LIN {X 0,Y 382.363,Z 610.569,A -85,B 0,C 180,E1 -11975.801,E2 -11975.801} C_VEL
LIN {X 0,Y 382.259,Z 606.99,A -85,B 0,C 180,E1 -11977.393,E2 -11977.393} C_VEL
LIN {X 0,Y 382.264,Z 602.395,A -85,B 0,C 180,E1 -11978.989,E2 -11978.989} C_VEL
LIN {X 0,Y 382.468,Z 595.707,A -85,B 0,C 180,E1 -11980.855,E2 -11980.855} C_VEL
LIN {X 0,Y 382.818,Z 587.32,A -85,B 0,C 180,E1 -11982.726,E2 -11982.726} C_VEL
LIN {X 0,Y 383.476,Z 578.596,A -85,B 0,C 180,E1 -11984.323,E2 -11984.323} C_VEL
LIN {X 0,Y 384.358,Z 568.07,A -85,B 0,C 180,E1 -11985.917,E2 -11985.917} C_VEL
LIN {X 0,Y 385.396,Z 557.58,A -85,B 0,C 180,E1 -11987.236,E2 -11987.236} C_VEL
LIN {X 0,Y 386.433,Z 546.274,A -85,B 0,C 180,E1 -11988.42,E2 -11988.42} C_VEL
LIN {X 0,Y 387.509,Z 533.775,A -85,B 0,C 180,E1 -11989.493,E2 -11989.493} C_VEL
LIN {X 0,Y 387.828,Z 526.827,A -85,B 0,C 180,E1 -11990.006,E2 -11990.006} C_VEL
LIN {X 0,Y 386.566,Z 512.32,A -85,B 0,C 180,E1 -11990.954,E2 -11990.954} C_VEL
LIN {X 0,Y 384.765,Z 496.815,A -85,B 0,C 180,E1 -11991.736,E2 -11991.736} C_VEL
LIN {X 0,Y 383.032,Z 482.96,A -85,B 0,C 180,E1 -11992.27,E2 -11992.27} C_VEL
LIN {X 0,Y 383.628,Z 472.139,A -85,B 0,C 180,E1 -11995.499,E2 -11995.499} C_VEL
LIN {X 0,Y 384.429,Z 460.422,A -85,B 0,C 180,E1 -11999.048,E2 -11999.048} C_VEL
LIN {X 0,Y 385.201,Z 450.992,A -85,B 0,C 180,E1 -12001.943,E2 -12001.943} C_VEL
LIN {X 0,Y 386.105,Z 441.213,A -85,B 0,C 180,E1 -12005.005,E2 -12005.005} C_VEL
LIN {X 0,Y 387.399,Z 428.707,A -85,B 0,C 180,E1 -12009.008,E2 -12009.008} C_VEL
LIN {X 0,Y 387.577,Z 424.534,A -85,B 0,C 180,E1 -12010.395,E2 -12010.395} C_VEL
LIN {X 0,Y 386.394,Z 417.864,A -85,B 0,C 180,E1 -12012.764,E2 -12012.764} C_VEL
LIN {X 0,Y 384.278,Z 407.541,A -85,B 0,C 180,E1 -12016.612,E2 -12016.612} C_VEL
LIN {X 0,Y 383.036,Z 401.399,A -85,B 0,C 180,E1 -12019.079,E2 -12019.079} C_VEL
LIN {X 0,Y 382.99,Z 401.403,A -85,B 0,C 180,E1 -12022.731,E2 -12022.731} C_VEL
LIN {X 0,Y 383.008,Z 401.4,A -85,B 0,C 180,E1 -12025.659,E2 -12025.659} C_VEL
LIN {X 0,Y 382.977,Z 401.407,A -85,B 0,C 180,E1 -12029.081,E2 -12029.081} C_VEL
LIN {X 0,Y 383.047,Z 401.395,A -85,B 0,C 180,E1 -12032.698,E2 -12032.698} C_VEL
LIN {X 0,Y 383.023,Z 401.396,A -85,B 0,C 180,E1 -12036.192,E2 -12036.192} C_VEL
LIN {X 0,Y 383.045,Z 401.395,A -85,B 0,C 180,E1 -12039.598,E2 -12039.598} C_VEL
LIN {X 0,Y 383.094,Z 401.392,A -85,B 0,C 180,E1 -12042.931,E2 -12042.931} C_VEL
LIN {X 0,Y 383.115,Z 401.386,A -85,B 0,C 180,E1 -12046.463,E2 -12046.463} C_VEL
LIN {X 0,Y 383.13,Z 401.385,A -85,B 0,C 180,E1 -12049.43,E2 -12049.43} C_VEL
LIN {X 0,Y 383.262,Z 401.369,A -85,B 0,C 180,E1 -12052.625,E2 -12052.625} C_VEL
LIN {X 0,Y 383.19,Z 401.38,A -85,B 0,C 180,E1 -12054.739,E2 -12054.739} C_VEL
LIN {X 0,Y 383.378,Z 401.352,A -85,B 0,C 180,E1 -12057.899,E2 -12057.899} C_VEL
LIN {X 0,Y 383.511,Z 401.335,A -85,B 0,C 180,E1 -12060,E2 -12060} C_VEL
LIN {X 0,Y 383.244,Z 401.372,A -85,B 0,C 180,E1 -12063.154,E2 -12063.154} C_VEL
LIN {X 0,Y 383.259,Z 401.366,A -85,B 0,C 180,E1 -12066.645,E2 -12066.645} C_VEL
LIN {X 0,Y 383.25,Z 401.37,A -85,B 0,C 180,E1 -12068.436,E2 -12068.436} C_VEL
LIN {X 0,Y 383.099,Z 401.387,A -85,B 0,C 180,E1 -12071.642,E2 -12071.642} C_VEL
LIN {X 0,Y 383.103,Z 401.392,A -85,B 0,C 180,E1 -12074.882,E2 -12074.882} C_VEL
LIN {X 0,Y 383.08,Z 401.39,A -85,B 0,C 180,E1 -12078.173,E2 -12078.173} C_VEL
LIN {X 0,Y 382.984,Z 401.401,A -85,B 0,C 180,E1 -12081.532,E2 -12081.532} C_VEL
LIN {X 0,Y 383.044,Z 401.397,A -85,B 0,C 180,E1 -12084.961,E2 -12084.961} C_VEL
LIN {X 0,Y 383.032,Z 401.4,A -85,B 0,C 180,E1 -12088.494,E2 -12088.494} C_VEL
LIN {X 0,Y 383.001,Z 401.4,A -85,B 0,C 180,E1 -12092.151,E2 -12092.151} C_VEL
LIN {X 0,Y 383.011,Z 401.403,A -85,B 0,C 180,E1 -12094.669,E2 -12094.669} C_VEL
LIN {X 0,Y 382.995,Z 401.4,A -85,B 0,C 180,E1 -12097.906,E2 -12097.906} C_VEL
LIN {X 0,Y 382.979,Z 401.402,A -85,B 0,C 180,E1 -12101.349,E2 -12101.349} C_VEL
LIN {X 0,Y 382.993,Z 401.404,A -85,B 0,C 180,E1 -12104.305,E2 -12104.305} C_VEL
LIN {X 0,Y 383.035,Z 401.395,A -85,B 0,C 180,E1 -12107.246,E2 -12107.246} C_VEL
LIN {X 0,Y 383.018,Z 401.402,A -85,B 0,C 180,E1 -12110.414,E2 -12110.414} C_VEL
LIN {X 0,Y 383.024,Z 401.398,A -85,B 0,C 180,E1 -12114.046,E2 -12114.046} C_VEL
LIN {X 0,Y 382.985,Z 401.401,A -85,B 0,C 180,E1 -12117.579,E2 -12117.579} C_VEL
LIN {X 0,Y 382.991,Z 401.405,A -85,B 0,C 180,E1 -12120.302,E2 -12120.302} C_VEL
LIN {X 0,Y 383.08,Z 401.392,A -85,B 0,C 180,E1 -12124.022,E2 -12124.022} C_VEL
LIN {X 0,Y 383.009,Z 401.398,A -85,B 0,C 180,E1 -12127.337,E2 -12127.337} C_VEL
LIN {X 0,Y 383.061,Z 401.394,A -85,B 0,C 180,E1 -12130.718,E2 -12130.718} C_VEL
LIN {X 0,Y 383.097,Z 401.388,A -85,B 0,C 180,E1 -12132.932,E2 -12132.932} C_VEL
LIN {X 0,Y 383.012,Z 401.402,A -85,B 0,C 180,E1 -12134.47,E2 -12134.47} C_VEL
LIN {X 0,Y 387.985,Z 416.324,A -85,B 0,C 180,E1 -12135.256,E2 -12135.256} C_VEL
LIN {X 0,Y 389.085,Z 421.064,A -85,B 0,C 180,E1 -12135.54,E2 -12135.54} C_VEL
LIN {X 0,Y 388.565,Z 433.969,A -85,B 0,C 180,E1 -12136.315,E2 -12136.315} C_VEL
LIN {X 0,Y 388.044,Z 444.903,A -85,B 0,C 180,E1 -12137.183,E2 -12137.183} C_VEL
LIN {X 0,Y 387.333,Z 455.355,A -85,B 0,C 180,E1 -12138.223,E2 -12138.223} C_VEL
LIN {X 0,Y 386.486,Z 465.755,A -85,B 0,C 180,E1 -12139.524,E2 -12139.524} C_VEL
LIN {X 0,Y 385.692,Z 474.22,A -85,B 0,C 180,E1 -12140.827,E2 -12140.827} C_VEL
LIN {X 0,Y 385.01,Z 482.449,A -85,B 0,C 180,E1 -12142.396,E2 -12142.396} C_VEL
LIN {X 0,Y 384.369,Z 488.071,A -85,B 0,C 180,E1 -12143.703,E2 -12143.703} C_VEL
LIN {X 0,Y 383.98,Z 493.516,A -85,B 0,C 180,E1 -12145.277,E2 -12145.277} C_VEL
LIN {X 0,Y 383.57,Z 497.804,A -85,B 0,C 180,E1 -12146.85,E2 -12146.85} C_VEL
LIN {X 0,Y 383.338,Z 500.063,A -85,B 0,C 180,E1 -12147.9,E2 -12147.9} C_VEL
LIN {X 0,Y 383.162,Z 501.911,A -85,B 0,C 180,E1 -12148.95,E2 -12148.95} C_VEL
LIN {X 0,Y 383.063,Z 503.34,A -85,B 0,C 180,E1 -12150.001,E2 -12150.001} C_VEL
LIN {X 0,Y 382.952,Z 504.968,A -85,B 0,C 180,E1 -12152.105,E2 -12152.105} C_VEL
LIN {X 0,Y 382.814,Z 505.247,A -85,B 0,C 180,E1 -12153.158,E2 -12153.158} C_VEL
LIN {X 0,Y 382.896,Z 505.095,A -85,B 0,C 180,E1 -12154.212,E2 -12154.212} C_VEL
LIN {X 0,Y 383.317,Z 503.595,A -85,B 0,C 180,E1 -12156.317,E2 -12156.317} C_VEL
LIN {X 0,Y 383.415,Z 502.3,A -85,B 0,C 180,E1 -12157.373,E2 -12157.373} C_VEL
LIN {X 0,Y 383.763,Z 499.52,A -85,B 0,C 180,E1 -12158.956,E2 -12158.956} C_VEL
LIN {X 0,Y 384.263,Z 495.718,A -85,B 0,C 180,E1 -12160.539,E2 -12160.539} C_VEL
LIN {X 0,Y 384.845,Z 490.786,A -85,B 0,C 180,E1 -12162.124,E2 -12162.124} C_VEL
LIN {X 0,Y 385.454,Z 484.548,A -85,B 0,C 180,E1 -12163.712,E2 -12163.712} C_VEL
LIN {X 0,Y 386.105,Z 478.122,A -85,B 0,C 180,E1 -12165.045,E2 -12165.045} C_VEL
LIN {X 0,Y 387.097,Z 468.732,A -85,B 0,C 180,E1 -12166.617,E2 -12166.617} C_VEL
LIN {X 0,Y 387.968,Z 458.877,A -85,B 0,C 180,E1 -12167.937,E2 -12167.937} C_VEL
LIN {X 0,Y 388.777,Z 447.77,A -85,B 0,C 180,E1 -12169.125,E2 -12169.125} C_VEL
LIN {X 0,Y 389.444,Z 436.792,A -85,B 0,C 180,E1 -12170.053,E2 -12170.053} C_VEL
LIN {X 0,Y 390.008,Z 425.18,A -85,B 0,C 180,E1 -12170.803,E2 -12170.803} C_VEL
LIN {X 0,Y 390.107,Z 422.244,A -85,B 0,C 180,E1 -12170.963,E2 -12170.963} C_VEL
LIN {X 0,Y 388.328,Z 416.045,A -85,B 0,C 180,E1 -12171.374,E2 -12171.374} C_VEL
LIN {X 0,Y 387.071,Z 414.332,A -85,B 0,C 180,E1 -12171.523,E2 -12171.523} C_VEL
LIN {X 0,Y 383.658,Z 412.795,A -85,B 0,C 180,E1 -12171.79,E2 -12171.79} C_VEL
LIN {X 0,Y 379.835,Z 411.072,A -85,B 0,C 180,E1 -12172.082,E2 -12172.082} C_VEL
LIN {X 0,Y 378.709,Z 409.608,A -85,B 0,C 180,E1 -12172.201,E2 -12172.201} C_VEL
LIN {X 0,Y 376.021,Z 402.772,A -85,B 0,C 180,E1 -12172.57,E2 -12172.57} C_VEL
LIN {X 0,Y 375.946,Z 402.28,A -85,B 0,C 180,E1 -12172.628,E2 -12172.628} C_VEL
LIN {X 0,Y 376.048,Z 402.268,A -85,B 0,C 180,E1 -12176.222,E2 -12176.222} C_VEL
LIN {X 0,Y 375.976,Z 402.279,A -85,B 0,C 180,E1 -12179.08,E2 -12179.08} C_VEL
LIN {X 0,Y 375.955,Z 402.283,A -85,B 0,C 180,E1 -12182.829,E2 -12182.829} C_VEL
LIN {X 0,Y 375.963,Z 402.28,A -85,B 0,C 180,E1 -12185.416,E2 -12185.416} C_VEL
LIN {X 0,Y 375.978,Z 402.264,A -85,B 0,C 180,E1 -12188.271,E2 -12188.271} C_VEL
LIN {X 0,Y 375.94,Z 402.28,A -85,B 0,C 180,E1 -12191.601,E2 -12191.601} C_VEL
LIN {X 0,Y 375.934,Z 402.277,A -85,B 0,C 180,E1 -12195.268,E2 -12195.268} C_VEL
LIN {X 0,Y 375.946,Z 402.278,A -85,B 0,C 180,E1 -12198.398,E2 -12198.398} C_VEL
LIN {X 0,Y 375.98,Z 402.25,A -85,B 0,C 180,E1 -12201.729,E2 -12201.729} C_VEL
LIN {X 0,Y 375.985,Z 402.274,A -85,B 0,C 180,E1 -12205.333,E2 -12205.333} C_VEL
LIN {X 0,Y 375.962,Z 402.26,A -85,B 0,C 180,E1 -12208.438,E2 -12208.438} C_VEL
LIN {X 0,Y 375.988,Z 402.254,A -85,B 0,C 180,E1 -12212.14,E2 -12212.14} C_VEL
LIN {X 0,Y 376.01,Z 402.27,A -85,B 0,C 180,E1 -12214.539,E2 -12214.539} C_VEL
LIN {X 0,Y 375.961,Z 402.28,A -85,B 0,C 180,E1 -12218.045,E2 -12218.045} C_VEL
LIN {X 0,Y 376.023,Z 402.297,A -85,B 0,C 180,E1 -12219.949,E2 -12219.949} C_VEL
LIN {X 0,Y 379.982,Z 415.54,A -85,B 0,C 180,E1 -12221.014,E2 -12221.014} C_VEL
LIN {X 0,Y 382.285,Z 423.976,A -85,B 0,C 180,E1 -12221.788,E2 -12221.788} C_VEL
LIN {X 0,Y 381.339,Z 437.114,A -85,B 0,C 180,E1 -12222.988,E2 -12222.988} C_VEL
LIN {X 0,Y 380.375,Z 449.046,A -85,B 0,C 180,E1 -12224.322,E2 -12224.322} C_VEL
LIN {X 0,Y 379.372,Z 459.947,A -85,B 0,C 180,E1 -12225.791,E2 -12225.791} C_VEL
LIN {X 0,Y 378.47,Z 469.862,A -85,B 0,C 180,E1 -12227.397,E2 -12227.397} C_VEL
LIN {X 0,Y 377.83,Z 478.131,A -85,B 0,C 180,E1 -12229.008,E2 -12229.008} C_VEL
LIN {X 0,Y 377.23,Z 485.272,A -85,B 0,C 180,E1 -12230.672,E2 -12230.672} C_VEL
LIN {X 0,Y 376.743,Z 491.71,A -85,B 0,C 180,E1 -12232.496,E2 -12232.496} C_VEL
LIN {X 0,Y 376.436,Z 496.315,A -85,B 0,C 180,E1 -12234.106,E2 -12234.106} C_VEL
LIN {X 0,Y 376.011,Z 500.074,A -85,B 0,C 180,E1 -12235.712,E2 -12235.712} C_VEL
LIN {X 0,Y 375.95,Z 503.669,A -85,B 0,C 180,E1 -12237.857,E2 -12237.857} C_VEL
LIN {X 0,Y 375.983,Z 505.886,A -85,B 0,C 180,E1 -12240,E2 -12240} C_VEL
LIN {X 0,Y 376.156,Z 506.754,A -85,B 0,C 180,E1 -12242.141,E2 -12242.141} C_VEL
LIN {X 0,Y 376.352,Z 506.311,A -85,B 0,C 180,E1 -12244.284,E2 -12244.284} C_VEL
LIN {X 0,Y 376.78,Z 504.524,A -85,B 0,C 180,E1 -12246.426,E2 -12246.426} C_VEL
LIN {X 0,Y 377.511,Z 501.315,A -85,B 0,C 180,E1 -12248.565,E2 -12248.565} C_VEL
LIN {X 0,Y 378.417,Z 496.588,A -85,B 0,C 180,E1 -12250.703,E2 -12250.703} C_VEL
LIN {X 0,Y 379.495,Z 490.27,A -85,B 0,C 180,E1 -12252.84,E2 -12252.84} C_VEL
LIN {X 0,Y 380.744,Z 483.181,A -85,B 0,C 180,E1 -12254.703,E2 -12254.703} C_VEL
LIN {X 0,Y 382.13,Z 475.231,A -85,B 0,C 180,E1 -12256.389,E2 -12256.389} C_VEL
LIN {X 0,Y 383.693,Z 465.133,A -85,B 0,C 180,E1 -12258.142,E2 -12258.142} C_VEL
LIN {X 0,Y 385.278,Z 453.986,A -85,B 0,C 180,E1 -12259.722,E2 -12259.722} C_VEL
LIN {X 0,Y 386.757,Z 442.713,A -85,B 0,C 180,E1 -12261.032,E2 -12261.032} C_VEL
LIN {X 0,Y 387.957,Z 430.591,A -85,B 0,C 180,E1 -12262.205,E2 -12262.205} C_VEL
LIN {X 0,Y 384.234,Z 419.734,A -85,B 0,C 180,E1 -12263.593,E2 -12263.593} C_VEL
LIN {X 0,Y 379.672,Z 409.782,A -85,B 0,C 180,E1 -12264.901,E2 -12264.901} C_VEL
LIN {X 0,Y 376.274,Z 403.382,A -85,B 0,C 180,E1 -12265.767,E2 -12265.767} C_VEL
LIN {X 0,Y 376.052,Z 402.271,A -85,B 0,C 180,E1 -12265.892,E2 -12265.892} C_VEL
LIN {X 0,Y 375.964,Z 402.278,A -85,B 0,C 180,E1 -12269.079,E2 -12269.079} C_VEL
LIN {X 0,Y 375.952,Z 402.283,A -85,B 0,C 180,E1 -12272.828,E2 -12272.828} C_VEL
LIN {X 0,Y 375.96,Z 402.279,A -85,B 0,C 180,E1 -12275.415,E2 -12275.415} C_VEL
LIN {X 0,Y 375.977,Z 402.408,A -85,B 0,C 180,E1 -12278.27,E2 -12278.27} C_VEL
LIN {X 0,Y 376.57,Z 405.287,A -85,B 0,C 180,E1 -12280.784,E2 -12280.784} C_VEL
LIN {X 0,Y 377.707,Z 410.283,A -85,B 0,C 180,E1 -12284.248,E2 -12284.248} C_VEL
LIN {X 0,Y 378.756,Z 415.501,A -85,B 0,C 180,E1 -12287.157,E2 -12287.157} C_VEL
LIN {X 0,Y 379.674,Z 420.677,A -85,B 0,C 180,E1 -12289.618,E2 -12289.618} C_VEL
LIN {X 0,Y 379.475,Z 424.001,A -85,B 0,C 180,E1 -12290.972,E2 -12290.972} C_VEL
LIN {X 0,Y 377.905,Z 434.883,A -85,B 0,C 180,E1 -12294.913,E2 -12294.913} C_VEL
LIN {X 0,Y 377.182,Z 443.913,A -85,B 0,C 180,E1 -12297.923,E2 -12297.923} C_VEL
LIN {X 0,Y 376.583,Z 453.62,A -85,B 0,C 180,E1 -12300.972,E2 -12300.972} C_VEL
LIN {X 0,Y 376.035,Z 465.666,A -85,B 0,C 180,E1 -12304.571,E2 -12304.571} C_VEL
LIN {X 0,Y 377.009,Z 470.108,A -85,B 0,C 180,E1 -12304.866,E2 -12304.866} C_VEL
LIN {X 0,Y 379.843,Z 484.021,A -85,B 0,C 180,E1 -12305.812,E2 -12305.812} C_VEL
LIN {X 0,Y 381.705,Z 498.234,A -85,B 0,C 180,E1 -12306.801,E2 -12306.801} C_VEL
LIN {X 0,Y 382.113,Z 512.565,A -85,B 0,C 180,E1 -12307.835,E2 -12307.835} C_VEL
LIN {X 0,Y 381.875,Z 526.325,A -85,B 0,C 180,E1 -12308.968,E2 -12308.968} C_VEL
LIN {X 0,Y 381.81,Z 532.357,A -85,B 0,C 180,E1 -12309.528,E2 -12309.528} C_VEL
LIN {X 0,Y 379.923,Z 546.761,A -85,B 0,C 180,E1 -12310.971,E2 -12310.971} C_VEL
LIN {X 0,Y 378.473,Z 558.846,A -85,B 0,C 180,E1 -12312.436,E2 -12312.436} C_VEL
LIN {X 0,Y 377.222,Z 570.003,A -85,B 0,C 180,E1 -12314.049,E2 -12314.049} C_VEL
LIN {X 0,Y 376.213,Z 580.893,A -85,B 0,C 180,E1 -12315.944,E2 -12315.944} C_VEL
LIN {X 0,Y 375.542,Z 589.889,A -85,B 0,C 180,E1 -12317.845,E2 -12317.845} C_VEL
LIN {X 0,Y 375.22,Z 597.309,A -85,B 0,C 180,E1 -12319.749,E2 -12319.749} C_VEL
LIN {X 0,Y 375.164,Z 602.57,A -85,B 0,C 180,E1 -12321.38,E2 -12321.38} C_VEL
LIN {X 0,Y 375.265,Z 608.03,A -85,B 0,C 180,E1 -12323.547,E2 -12323.547} C_VEL
LIN {X 0,Y 375.506,Z 611.899,A -85,B 0,C 180,E1 -12325.705,E2 -12325.705} C_VEL
LIN {X 0,Y 375.511,Z 614.201,A -85,B 0,C 180,E1 -12327.854,E2 -12327.854} C_VEL
LIN {X 0,Y 375.691,Z 614.818,A -85,B 0,C 180,E1 -12328.927,E2 -12328.927} C_VEL
LIN {X 0,Y 375.825,Z 615.054,A -85,B 0,C 180,E1 -12329.999,E2 -12329.999} C_VEL
LIN {X 0,Y 375.501,Z 614.309,A -85,B 0,C 180,E1 -12332.144,E2 -12332.144} C_VEL
LIN {X 0,Y 375.434,Z 612.09,A -85,B 0,C 180,E1 -12334.293,E2 -12334.293} C_VEL
LIN {X 0,Y 375.327,Z 609.351,A -85,B 0,C 180,E1 -12335.91,E2 -12335.91} C_VEL
LIN {X 0,Y 375.227,Z 605.712,A -85,B 0,C 180,E1 -12337.532,E2 -12337.532} C_VEL
LIN {X 0,Y 375.231,Z 601.088,A -85,B 0,C 180,E1 -12339.159,E2 -12339.159} C_VEL
LIN {X 0,Y 375.45,Z 594.312,A -85,B 0,C 180,E1 -12341.061,E2 -12341.061} C_VEL
LIN {X 0,Y 375.812,Z 585.811,A -85,B 0,C 180,E1 -12342.967,E2 -12342.967} C_VEL
LIN {X 0,Y 376.501,Z 576.99,A -85,B 0,C 180,E1 -12344.594,E2 -12344.594} C_VEL
LIN {X 0,Y 377.396,Z 566.348,A -85,B 0,C 180,E1 -12346.219,E2 -12346.219} C_VEL
LIN {X 0,Y 378.615,Z 554.584,A -85,B 0,C 180,E1 -12347.694,E2 -12347.694} C_VEL
LIN {X 0,Y 379.76,Z 542.914,A -85,B 0,C 180,E1 -12348.895,E2 -12348.895} C_VEL
LIN {X 0,Y 380.837,Z 530.246,A -85,B 0,C 180,E1 -12349.96,E2 -12349.96} C_VEL
LIN {X 0,Y 380.057,Z 517.099,A -85,B 0,C 180,E1 -12350.898,E2 -12350.898} C_VEL
LIN {X 0,Y 378.414,Z 501.733,A -85,B 0,C 180,E1 -12351.781,E2 -12351.781} C_VEL
LIN {X 0,Y 376.497,Z 486.522,A -85,B 0,C 180,E1 -12352.439,E2 -12352.439} C_VEL
LIN {X 0,Y 375.998,Z 482.128,A -85,B 0,C 180,E1 -12352.602,E2 -12352.602} C_VEL
LIN {X 0,Y 376.651,Z 471.246,A -85,B 0,C 180,E1 -12355.925,E2 -12355.925} C_VEL
LIN {X 0,Y 377.473,Z 459.49,A -85,B 0,C 180,E1 -12359.562,E2 -12359.562} C_VEL
LIN {X 0,Y 378.312,Z 449.87,A -85,B 0,C 180,E1 -12362.596,E2 -12362.596} C_VEL
LIN {X 0,Y 379.126,Z 441.262,A -85,B 0,C 180,E1 -12365.349,E2 -12365.349} C_VEL
LIN {X 0,Y 380.412,Z 429.764,A -85,B 0,C 180,E1 -12369.11,E2 -12369.11} C_VEL
LIN {X 0,Y 380.647,Z 426.345,A -85,B 0,C 180,E1 -12370.255,E2 -12370.255} C_VEL
LIN {X 0,Y 379.775,Z 420.772,A -85,B 0,C 180,E1 -12372.249,E2 -12372.249} C_VEL
LIN {X 0,Y 377.838,Z 411.394,A -85,B 0,C 180,E1 -12375.772,E2 -12375.772} C_VEL
LIN {X 0,Y 376.006,Z 402.275,A -85,B 0,C 180,E1 -12379.388,E2 -12379.388} C_VEL
LIN {X 0,Y 375.96,Z 402.281,A -85,B 0,C 180,E1 -12381.911,E2 -12381.911} C_VEL
LIN {X 0,Y 375.971,Z 402.279,A -85,B 0,C 180,E1 -12385.332,E2 -12385.332} C_VEL
LIN {X 0,Y 375.95,Z 402.277,A -85,B 0,C 180,E1 -12388.438,E2 -12388.438} C_VEL
LIN {X 0,Y 375.992,Z 402.271,A -85,B 0,C 180,E1 -12392.141,E2 -12392.141} C_VEL
LIN {X 0,Y 375.996,Z 402.272,A -85,B 0,C 180,E1 -12394.538,E2 -12394.538} C_VEL
LIN {X 0,Y 375.953,Z 402.276,A -85,B 0,C 180,E1 -12398.045,E2 -12398.045} C_VEL
LIN {X 0,Y 375.998,Z 402.273,A -85,B 0,C 180,E1 -12401.473,E2 -12401.473} C_VEL
LIN {X 0,Y 376.049,Z 402.269,A -85,B 0,C 180,E1 -12404.832,E2 -12404.832} C_VEL
LIN {X 0,Y 376.048,Z 402.265,A -85,B 0,C 180,E1 -12408.137,E2 -12408.137} C_VEL
LIN {X 0,Y 376.247,Z 402.24,A -85,B 0,C 180,E1 -12411.877,E2 -12411.877} C_VEL
LIN {X 0,Y 376.162,Z 402.254,A -85,B 0,C 180,E1 -12414.64,E2 -12414.64} C_VEL
LIN {X 0,Y 376.344,Z 402.228,A -85,B 0,C 180,E1 -12417.86,E2 -12417.86} C_VEL
LIN {X 0,Y 376.48,Z 402.211,A -85,B 0,C 180,E1 -12420,E2 -12420} C_VEL
LIN {X 0,Y 376.182,Z 402.251,A -85,B 0,C 180,E1 -12423.213,E2 -12423.213} C_VEL
LIN {X 0,Y 376.224,Z 402.243,A -85,B 0,C 180,E1 -12426.636,E2 -12426.636} C_VEL
LIN {X 0,Y 376.196,Z 402.25,A -85,B 0,C 180,E1 -12428.596,E2 -12428.596} C_VEL
LIN {X 0,Y 376.05,Z 402.264,A -85,B 0,C 180,E1 -12431.864,E2 -12431.864} C_VEL
LIN {X 0,Y 376.05,Z 402.267,A -85,B 0,C 180,E1 -12435.168,E2 -12435.168} C_VEL
LIN {X 0,Y 376.014,Z 402.273,A -85,B 0,C 180,E1 -12438.527,E2 -12438.527} C_VEL
LIN {X 0,Y 375.954,Z 402.277,A -85,B 0,C 180,E1 -12441.955,E2 -12441.955} C_VEL
LIN {X 0,Y 375.997,Z 402.271,A -85,B 0,C 180,E1 -12445.462,E2 -12445.462} C_VEL
LIN {X 0,Y 375.962,Z 402.278,A -85,B 0,C 180,E1 -12449.08,E2 -12449.08} C_VEL
LIN {X 0,Y 375.941,Z 402.282,A -85,B 0,C 180,E1 -12452.83,E2 -12452.83} C_VEL
LIN {X 0,Y 375.951,Z 402.277,A -85,B 0,C 180,E1 -12455.417,E2 -12455.417} C_VEL
LIN {X 0,Y 375.97,Z 402.278,A -85,B 0,C 180,E1 -12458.272,E2 -12458.272} C_VEL
LIN {X 0,Y 375.93,Z 402.279,A -85,B 0,C 180,E1 -12461.602,E2 -12461.602} C_VEL
LIN {X 0,Y 375.924,Z 402.28,A -85,B 0,C 180,E1 -12465.27,E2 -12465.27} C_VEL
LIN {X 0,Y 375.957,Z 402.281,A -85,B 0,C 180,E1 -12468.396,E2 -12468.396} C_VEL
LIN {X 0,Y 375.975,Z 402.274,A -85,B 0,C 180,E1 -12471.73,E2 -12471.73} C_VEL
LIN {X 0,Y 375.977,Z 402.273,A -85,B 0,C 180,E1 -12475.334,E2 -12475.334} C_VEL
LIN {X 0,Y 375.956,Z 402.282,A -85,B 0,C 180,E1 -12478.44,E2 -12478.44} C_VEL
LIN {X 0,Y 375.982,Z 402.277,A -85,B 0,C 180,E1 -12482.142,E2 -12482.142} C_VEL
LIN {X 0,Y 376.006,Z 402.274,A -85,B 0,C 180,E1 -12484.541,E2 -12484.541} C_VEL
LIN {X 0,Y 375.964,Z 402.279,A -85,B 0,C 180,E1 -12488.047,E2 -12488.047} C_VEL
LIN {X 0,Y 376.009,Z 402.27,A -85,B 0,C 180,E1 -12491.475,E2 -12491.475} C_VEL
LIN {X 0,Y 375.996,Z 402.393,A -85,B 0,C 180,E1 -12494.16,E2 -12494.16} C_VEL
LIN {X 0,Y 380.292,Z 414.972,A -85,B 0,C 180,E1 -12494.805,E2 -12494.805} C_VEL
LIN {X 0,Y 382.114,Z 420.87,A -85,B 0,C 180,E1 -12495.174,E2 -12495.174} C_VEL
LIN {X 0,Y 382.131,Z 427.467,A -85,B 0,C 180,E1 -12495.543,E2 -12495.543} C_VEL
LIN {X 0,Y 381.551,Z 440.065,A -85,B 0,C 180,E1 -12496.419,E2 -12496.419} C_VEL
LIN {X 0,Y 380.868,Z 451.755,A -85,B 0,C 180,E1 -12497.479,E2 -12497.479} C_VEL
LIN {X 0,Y 380.077,Z 461.602,A -85,B 0,C 180,E1 -12498.606,E2 -12498.606} C_VEL
LIN {X 0,Y 379.29,Z 470.557,A -85,B 0,C 180,E1 -12499.863,E2 -12499.863} C_VEL
LIN {X 0,Y 378.594,Z 478.328,A -85,B 0,C 180,E1 -12501.192,E2 -12501.192} C_VEL
LIN {X 0,Y 377.81,Z 485.965,A -85,B 0,C 180,E1 -12502.788,E2 -12502.788} C_VEL
LIN {X 0,Y 377.314,Z 491.123,A -85,B 0,C 180,E1 -12504.121,E2 -12504.121} C_VEL
LIN {X 0,Y 376.859,Z 496.162,A -85,B 0,C 180,E1 -12505.723,E2 -12505.723} C_VEL
LIN {X 0,Y 376.483,Z 500.069,A -85,B 0,C 180,E1 -12507.326,E2 -12507.326} C_VEL
LIN {X 0,Y 376.142,Z 502.97,A -85,B 0,C 180,E1 -12508.931,E2 -12508.931} C_VEL
LIN {X 0,Y 376.042,Z 504.379,A -85,B 0,C 180,E1 -12510.001,E2 -12510.001} C_VEL
LIN {X 0,Y 375.928,Z 505.988,A -85,B 0,C 180,E1 -12512.144,E2 -12512.144} C_VEL
LIN {X 0,Y 375.79,Z 506.257,A -85,B 0,C 180,E1 -12513.217,E2 -12513.217} C_VEL
LIN {X 0,Y 376.042,Z 505.517,A -85,B 0,C 180,E1 -12515.363,E2 -12515.363} C_VEL
LIN {X 0,Y 376.325,Z 504.564,A -85,B 0,C 180,E1 -12516.435,E2 -12516.435} C_VEL
LIN {X 0,Y 376.433,Z 503.254,A -85,B 0,C 180,E1 -12517.511,E2 -12517.511} C_VEL
LIN {X 0,Y 376.818,Z 500.452,A -85,B 0,C 180,E1 -12519.123,E2 -12519.123} C_VEL
LIN {X 0,Y 377.341,Z 496.627,A -85,B 0,C 180,E1 -12520.735,E2 -12520.735} C_VEL
LIN {X 0,Y 377.958,Z 491.663,A -85,B 0,C 180,E1 -12522.348,E2 -12522.348} C_VEL
LIN {X 0,Y 378.585,Z 485.397,A -85,B 0,C 180,E1 -12523.966,E2 -12523.966} C_VEL
LIN {X 0,Y 379.296,Z 479.016,A -85,B 0,C 180,E1 -12525.306,E2 -12525.306} C_VEL
LIN {X 0,Y 380.349,Z 469.506,A -85,B 0,C 180,E1 -12526.92,E2 -12526.92} C_VEL
LIN {X 0,Y 381.265,Z 459.578,A -85,B 0,C 180,E1 -12528.263,E2 -12528.263} C_VEL
LIN {X 0,Y 382.104,Z 448.455,A -85,B 0,C 180,E1 -12529.468,E2 -12529.468} C_VEL
LIN {X 0,Y 382.823,Z 437.305,A -85,B 0,C 180,E1 -12530.415,E2 -12530.415} C_VEL
LIN {X 0,Y 383.423,Z 424.433,A -85,B 0,C 180,E1 -12531.24,E2 -12531.24} C_VEL
LIN {X 0,Y 383.066,Z 422.118,A -85,B 0,C 180,E1 -12531.392,E2 -12531.392} C_VEL
LIN {X 0,Y 379.018,Z 410.536,A -85,B 0,C 180,E1 -12532.15,E2 -12532.15} C_VEL
LIN {X 0,Y 378.709,Z 409.608,A -85,B 0,C 180,E1 -12532.201,E2 -12532.201} C_VEL
LIN {X 0,Y 377.218,Z 406.796,A -85,B 0,C 180,E1 -12532.493,E2 -12532.493} C_VEL
LIN {X 0,Y 375.573,Z 404.854,A -85,B 0,C 180,E1 -12532.918,E2 -12532.918} C_VEL
LIN {X 0,Y 373.173,Z 403.244,A -85,B 0,C 180,E1 -12533.699,E2 -12533.699} C_VEL
LIN {X 0,Y 371.095,Z 402.885,A -85,B 0,C 180,E1 -12534.607,E2 -12534.607} C_VEL
LIN {X 0,Y 369.268,Z 403.118,A -85,B 0,C 180,E1 -12535.91,E2 -12535.91} C_VEL
LIN {X 0,Y 368.982,Z 403.149,A -85,B 0,C 180,E1 -12536.577,E2 -12536.577} C_VEL
LIN {X 0,Y 368.925,Z 403.157,A -85,B 0,C 180,E1 -12539.69,E2 -12539.69} C_VEL
LIN {X 0,Y 368.903,Z 403.162,A -85,B 0,C 180,E1 -12543.044,E2 -12543.044} C_VEL
LIN {X 0,Y 368.923,Z 403.159,A -85,B 0,C 180,E1 -12546.197,E2 -12546.197} C_VEL
LIN {X 0,Y 368.908,Z 403.147,A -85,B 0,C 180,E1 -12548.954,E2 -12548.954} C_VEL
LIN {X 0,Y 368.887,Z 403.159,A -85,B 0,C 180,E1 -12552.01,E2 -12552.01} C_VEL
LIN {X 0,Y 368.887,Z 403.155,A -85,B 0,C 180,E1 -12555.176,E2 -12555.176} C_VEL
LIN {X 0,Y 368.894,Z 403.159,A -85,B 0,C 180,E1 -12558.179,E2 -12558.179} C_VEL
LIN {X 0,Y 368.914,Z 403.128,A -85,B 0,C 180,E1 -12561.36,E2 -12561.36} C_VEL
LIN {X 0,Y 368.942,Z 403.151,A -85,B 0,C 180,E1 -12565.147,E2 -12565.147} C_VEL
LIN {X 0,Y 368.934,Z 403.129,A -85,B 0,C 180,E1 -12569.046,E2 -12569.046} C_VEL
LIN {X 0,Y 368.968,Z 403.136,A -85,B 0,C 180,E1 -12572.796,E2 -12572.796} C_VEL
LIN {X 0,Y 368.938,Z 403.154,A -85,B 0,C 180,E1 -12576.117,E2 -12576.117} C_VEL
LIN {X 0,Y 369,Z 403.222,A -85,B 0,C 180,E1 -12579.652,E2 -12579.652} C_VEL
LIN {X 0,Y 373.136,Z 417.093,A -85,B 0,C 180,E1 -12580.8,E2 -12580.8} C_VEL
LIN {X 0,Y 375.422,Z 425.391,A -85,B 0,C 180,E1 -12581.584,E2 -12581.584} C_VEL
LIN {X 0,Y 374.437,Z 438.415,A -85,B 0,C 180,E1 -12582.805,E2 -12582.805} C_VEL
LIN {X 0,Y 373.446,Z 450.377,A -85,B 0,C 180,E1 -12584.174,E2 -12584.174} C_VEL
LIN {X 0,Y 372.3,Z 462.078,A -85,B 0,C 180,E1 -12585.794,E2 -12585.794} C_VEL
LIN {X 0,Y 371.458,Z 471.828,A -85,B 0,C 180,E1 -12587.433,E2 -12587.433} C_VEL
LIN {X 0,Y 370.768,Z 479.963,A -85,B 0,C 180,E1 -12589.073,E2 -12589.073} C_VEL
LIN {X 0,Y 370.126,Z 487.468,A -85,B 0,C 180,E1 -12590.892,E2 -12590.892} C_VEL
LIN {X 0,Y 369.672,Z 494.136,A -85,B 0,C 180,E1 -12592.901,E2 -12592.901} C_VEL
LIN {X 0,Y 369.236,Z 499.736,A -85,B 0,C 180,E1 -12595.086,E2 -12595.086} C_VEL
LIN {X 0,Y 368.848,Z 502.991,A -85,B 0,C 180,E1 -12596.723,E2 -12596.723} C_VEL
LIN {X 0,Y 368.933,Z 505.958,A -85,B 0,C 180,E1 -12598.908,E2 -12598.908} C_VEL
LIN {X 0,Y 369.028,Z 507.584,A -85,B 0,C 180,E1 -12601.091,E2 -12601.091} C_VEL
LIN {X 0,Y 369.279,Z 507.87,A -85,B 0,C 180,E1 -12603.273,E2 -12603.273} C_VEL
LIN {X 0,Y 369.582,Z 506.84,A -85,B 0,C 180,E1 -12605.456,E2 -12605.456} C_VEL
LIN {X 0,Y 370.228,Z 504.44,A -85,B 0,C 180,E1 -12607.636,E2 -12607.636} C_VEL
LIN {X 0,Y 371.145,Z 500.612,A -85,B 0,C 180,E1 -12609.812,E2 -12609.812} C_VEL
LIN {X 0,Y 372.153,Z 495.213,A -85,B 0,C 180,E1 -12611.989,E2 -12611.989} C_VEL
LIN {X 0,Y 373.146,Z 490.052,A -85,B 0,C 180,E1 -12613.617,E2 -12613.617} C_VEL
LIN {X 0,Y 374.539,Z 482.629,A -85,B 0,C 180,E1 -12615.509,E2 -12615.509} C_VEL
LIN {X 0,Y 376.207,Z 473.451,A -85,B 0,C 180,E1 -12617.391,E2 -12617.391} C_VEL
LIN {X 0,Y 377.789,Z 463.884,A -85,B 0,C 180,E1 -12618.999,E2 -12618.999} C_VEL
LIN {X 0,Y 379.374,Z 453.319,A -85,B 0,C 180,E1 -12620.467,E2 -12620.467} C_VEL
LIN {X 0,Y 381.15,Z 440.629,A -85,B 0,C 180,E1 -12621.894,E2 -12621.894} C_VEL
LIN {X 0,Y 381.945,Z 433.385,A -85,B 0,C 180,E1 -12622.598,E2 -12622.598} C_VEL
LIN {X 0,Y 378.128,Z 422.086,A -85,B 0,C 180,E1 -12624.135,E2 -12624.135} C_VEL
LIN {X 0,Y 373.099,Z 411.187,A -85,B 0,C 180,E1 -12625.674,E2 -12625.674} C_VEL
LIN {X 0,Y 370.614,Z 406.842,A -85,B 0,C 180,E1 -12626.339,E2 -12626.339} C_VEL
LIN {X 0,Y 369.496,Z 405.037,A -85,B 0,C 180,E1 -12626.623,E2 -12626.623} C_VEL
LIN {X 0,Y 368.961,Z 403.154,A -85,B 0,C 180,E1 -12626.857,E2 -12626.857} C_VEL
LIN {X 0,Y 368.918,Z 403.158,A -85,B 0,C 180,E1 -12629.69,E2 -12629.69} C_VEL
LIN {X 0,Y 368.9,Z 403.159,A -85,B 0,C 180,E1 -12633.043,E2 -12633.043} C_VEL
LIN {X 0,Y 368.943,Z 403.153,A -85,B 0,C 180,E1 -12636.523,E2 -12636.523} C_VEL
LIN {X 0,Y 369.045,Z 403.869,A -85,B 0,C 180,E1 -12637.546,E2 -12637.546} C_VEL
LIN {X 0,Y 369.748,Z 407.086,A -85,B 0,C 180,E1 -12640.508,E2 -12640.508} C_VEL
LIN {X 0,Y 370.803,Z 411.85,A -85,B 0,C 180,E1 -12643.925,E2 -12643.925} C_VEL
LIN {X 0,Y 371.929,Z 417.444,A -85,B 0,C 180,E1 -12647.135,E2 -12647.135} C_VEL
LIN {X 0,Y 372.803,Z 422.467,A -85,B 0,C 180,E1 -12649.574,E2 -12649.574} C_VEL
LIN {X 0,Y 372.462,Z 426.041,A -85,B 0,C 180,E1 -12651.05,E2 -12651.05} C_VEL
LIN {X 0,Y 370.835,Z 437.71,A -85,B 0,C 180,E1 -12655.35,E2 -12655.35} C_VEL
LIN {X 0,Y 369.922,Z 448.994,A -85,B 0,C 180,E1 -12659.138,E2 -12659.138} C_VEL
LIN {X 0,Y 369.222,Z 460.701,A -85,B 0,C 180,E1 -12662.816,E2 -12662.816} C_VEL
LIN {X 0,Y 369.117,Z 463.524,A -85,B 0,C 180,E1 -12663.674,E2 -12663.674} C_VEL
LIN {X 0,Y 370.16,Z 468.179,A -85,B 0,C 180,E1 -12664.021,E2 -12664.021} C_VEL
LIN {X 0,Y 373.247,Z 482.636,A -85,B 0,C 180,E1 -12665.095,E2 -12665.095} C_VEL
LIN {X 0,Y 375.234,Z 498.186,A -85,B 0,C 180,E1 -12666.253,E2 -12666.253} C_VEL
LIN {X 0,Y 375.634,Z 511.67,A -85,B 0,C 180,E1 -12667.285,E2 -12667.285} C_VEL
LIN {X 0,Y 375.217,Z 526.679,A -85,B 0,C 180,E1 -12668.576,E2 -12668.576} C_VEL
LIN {X 0,Y 374.947,Z 534.034,A -85,B 0,C 180,E1 -12669.294,E2 -12669.294} C_VEL
LIN {X 0,Y 373.014,Z 547.786,A -85,B 0,C 180,E1 -12670.747,E2 -12670.747} C_VEL
LIN {X 0,Y 371.4,Z 560.388,A -85,B 0,C 180,E1 -12672.375,E2 -12672.375} C_VEL
LIN {X 0,Y 370.13,Z 571.049,A -85,B 0,C 180,E1 -12674.018,E2 -12674.018} C_VEL
LIN {X 0,Y 369.097,Z 581.688,A -85,B 0,C 180,E1 -12675.985,E2 -12675.985} C_VEL
LIN {X 0,Y 368.436,Z 590.195,A -85,B 0,C 180,E1 -12677.887,E2 -12677.887} C_VEL
LIN {X 0,Y 368.172,Z 596.401,A -85,B 0,C 180,E1 -12679.551,E2 -12679.551} C_VEL
LIN {X 0,Y 368.104,Z 603.111,A -85,B 0,C 180,E1 -12681.766,E2 -12681.766} C_VEL
LIN {X 0,Y 368.203,Z 607.03,A -85,B 0,C 180,E1 -12683.423,E2 -12683.423} C_VEL
LIN {X 0,Y 368.466,Z 610.869,A -85,B 0,C 180,E1 -12685.623,E2 -12685.623} C_VEL
LIN {X 0,Y 368.478,Z 613.143,A -85,B 0,C 180,E1 -12687.813,E2 -12687.813} C_VEL
LIN {X 0,Y 368.671,Z 613.747,A -85,B 0,C 180,E1 -12688.907,E2 -12688.907} C_VEL
LIN {X 0,Y 368.819,Z 613.967,A -85,B 0,C 180,E1 -12689.999,E2 -12689.999} C_VEL
LIN {X 0,Y 368.479,Z 613.175,A -85,B 0,C 180,E1 -12692.185,E2 -12692.185} C_VEL
LIN {X 0,Y 368.403,Z 610.906,A -85,B 0,C 180,E1 -12694.375,E2 -12694.375} C_VEL
LIN {X 0,Y 368.292,Z 608.115,A -85,B 0,C 180,E1 -12696.023,E2 -12696.023} C_VEL
LIN {X 0,Y 368.168,Z 602.979,A -85,B 0,C 180,E1 -12698.23,E2 -12698.23} C_VEL
LIN {X 0,Y 368.198,Z 597.897,A -85,B 0,C 180,E1 -12699.89,E2 -12699.89} C_VEL
LIN {X 0,Y 368.512,Z 590.597,A -85,B 0,C 180,E1 -12701.829,E2 -12701.829} C_VEL
LIN {X 0,Y 369,Z 581.624,A -85,B 0,C 180,E1 -12703.749,E2 -12703.749} C_VEL
LIN {X 0,Y 369.812,Z 572.003,A -85,B 0,C 180,E1 -12705.428,E2 -12705.428} C_VEL
LIN {X 0,Y 370.921,Z 560.512,A -85,B 0,C 180,E1 -12707.077,E2 -12707.077} C_VEL
LIN {X 0,Y 372.048,Z 548.917,A -85,B 0,C 180,E1 -12708.444,E2 -12708.444} C_VEL
LIN {X 0,Y 373.159,Z 537.49,A -85,B 0,C 180,E1 -12709.555,E2 -12709.555} C_VEL
LIN {X 0,Y 373.889,Z 529.684,A -85,B 0,C 180,E1 -12710.204,E2 -12710.204} C_VEL
LIN {X 0,Y 372.986,Z 516.66,A -85,B 0,C 180,E1 -12711.165,E2 -12711.165} C_VEL
LIN {X 0,Y 371.401,Z 501.484,A -85,B 0,C 180,E1 -12712.062,E2 -12712.062} C_VEL
LIN {X 0,Y 369.454,Z 485.668,A -85,B 0,C 180,E1 -12712.77,E2 -12712.77} C_VEL
LIN {X 0,Y 369.006,Z 481.253,A -85,B 0,C 180,E1 -12712.943,E2 -12712.943} C_VEL
LIN {X 0,Y 369.713,Z 469.271,A -85,B 0,C 180,E1 -12716.692,E2 -12716.692} C_VEL
LIN {X 0,Y 370.559,Z 458.324,A -85,B 0,C 180,E1 -12720.17,E2 -12720.17} C_VEL
LIN {X 0,Y 371.485,Z 448.698,A -85,B 0,C 180,E1 -12723.272,E2 -12723.272} C_VEL
LIN {X 0,Y 372.427,Z 438.976,A -85,B 0,C 180,E1 -12726.47,E2 -12726.47} C_VEL
LIN {X 0,Y 373.632,Z 429.146,A -85,B 0,C 180,E1 -12729.755,E2 -12729.755} C_VEL
LIN {X 0,Y 373.348,Z 425.068,A -85,B 0,C 180,E1 -12731.21,E2 -12731.21} C_VEL
LIN {X 0,Y 371.628,Z 416.555,A -85,B 0,C 180,E1 -12734.402,E2 -12734.402} C_VEL
LIN {X 0,Y 369.888,Z 407.867,A -85,B 0,C 180,E1 -12737.815,E2 -12737.815} C_VEL
LIN {X 0,Y 368.946,Z 403.155,A -85,B 0,C 180,E1 -12739.814,E2 -12739.814} C_VEL
LIN {X 0,Y 368.91,Z 403.155,A -85,B 0,C 180,E1 -12743.803,E2 -12743.803} C_VEL
LIN {X 0,Y 368.888,Z 403.16,A -85,B 0,C 180,E1 -12746.956,E2 -12746.956} C_VEL
LIN {X 0,Y 368.914,Z 403.153,A -85,B 0,C 180,E1 -12750.31,E2 -12750.31} C_VEL
LIN {X 0,Y 368.972,Z 403.148,A -85,B 0,C 180,E1 -12753.535,E2 -12753.535} C_VEL
LIN {X 0,Y 368.956,Z 403.148,A -85,B 0,C 180,E1 -12756.421,E2 -12756.421} C_VEL
LIN {X 0,Y 368.926,Z 403.152,A -85,B 0,C 180,E1 -12759.947,E2 -12759.947} C_VEL
LIN {X 0,Y 368.965,Z 403.149,A -85,B 0,C 180,E1 -12763.398,E2 -12763.398} C_VEL
LIN {X 0,Y 369.049,Z 403.14,A -85,B 0,C 180,E1 -12766.79,E2 -12766.79} C_VEL
LIN {X 0,Y 369.062,Z 403.135,A -85,B 0,C 180,E1 -12770.132,E2 -12770.132} C_VEL
LIN {X 0,Y 369.177,Z 403.121,A -85,B 0,C 180,E1 -12772.342,E2 -12772.342} C_VEL
LIN {X 0,Y 369.135,Z 403.128,A -85,B 0,C 180,E1 -12774.538,E2 -12774.538} C_VEL
LIN {X 0,Y 369.309,Z 403.104,A -85,B 0,C 180,E1 -12777.819,E2 -12777.819} C_VEL
LIN {X 0,Y 369.45,Z 403.086,A -85,B 0,C 180,E1 -12780,E2 -12780} C_VEL
LIN {X 0,Y 369.309,Z 403.104,A -85,B 0,C 180,E1 -12782.182,E2 -12782.182} C_VEL
LIN {X 0,Y 369.194,Z 403.121,A -85,B 0,C 180,E1 -12786.624,E2 -12786.624} C_VEL
LIN {X 0,Y 369.129,Z 403.132,A -85,B 0,C 180,E1 -12788.761,E2 -12788.761} C_VEL
LIN {X 0,Y 369.004,Z 403.142,A -85,B 0,C 180,E1 -12792.094,E2 -12792.094} C_VEL
LIN {X 0,Y 368.989,Z 403.144,A -85,B 0,C 180,E1 -12795.466,E2 -12795.466} C_VEL
LIN {X 0,Y 368.973,Z 403.151,A -85,B 0,C 180,E1 -12798.894,E2 -12798.894} C_VEL
LIN {X 0,Y 368.923,Z 403.155,A -85,B 0,C 180,E1 -12802.396,E2 -12802.396} C_VEL
LIN {X 0,Y 368.991,Z 403.144,A -85,B 0,C 180,E1 -12805.981,E2 -12805.981} C_VEL
LIN {X 0,Y 368.953,Z 403.153,A -85,B 0,C 180,E1 -12808.813,E2 -12808.813} C_VEL
LIN {X 0,Y 368.89,Z 403.158,A -85,B 0,C 180,E1 -12812.239,E2 -12812.239} C_VEL
LIN {X 0,Y 368.922,Z 403.154,A -85,B 0,C 180,E1 -12815.003,E2 -12815.003} C_VEL
LIN {X 0,Y 368.905,Z 403.16,A -85,B 0,C 180,E1 -12818.642,E2 -12818.642} C_VEL
LIN {X 0,Y 368.876,Z 403.159,A -85,B 0,C 180,E1 -12822.011,E2 -12822.011} C_VEL
LIN {X 0,Y 368.881,Z 403.158,A -85,B 0,C 180,E1 -12825.178,E2 -12825.178} C_VEL
LIN {X 0,Y 368.906,Z 403.157,A -85,B 0,C 180,E1 -12828.183,E2 -12828.183} C_VEL
LIN {X 0,Y 368.91,Z 403.154,A -85,B 0,C 180,E1 -12831.36,E2 -12831.36} C_VEL
LIN {X 0,Y 368.934,Z 403.151,A -85,B 0,C 180,E1 -12835.148,E2 -12835.148} C_VEL
LIN {X 0,Y 368.927,Z 403.152,A -85,B 0,C 180,E1 -12839.048,E2 -12839.048} C_VEL
LIN {X 0,Y 368.962,Z 403.149,A -85,B 0,C 180,E1 -12842.798,E2 -12842.798} C_VEL
LIN {X 0,Y 368.945,Z 403.153,A -85,B 0,C 180,E1 -12846.114,E2 -12846.114} C_VEL
LIN {X 0,Y 368.937,Z 403.153,A -85,B 0,C 180,E1 -12849.949,E2 -12849.949} C_VEL
LIN {X 0,Y 368.992,Z 403.149,A -85,B 0,C 180,E1 -12852.259,E2 -12852.259} C_VEL
LIN {X 0,Y 368.942,Z 403.227,A -85,B 0,C 180,E1 -12853.807,E2 -12853.807} C_VEL
LIN {X 0,Y 373.355,Z 416.1,A -85,B 0,C 180,E1 -12854.484,E2 -12854.484} C_VEL
LIN {X 0,Y 375.373,Z 422.49,A -85,B 0,C 180,E1 -12854.898,E2 -12854.898} C_VEL
LIN {X 0,Y 375.319,Z 430.353,A -85,B 0,C 180,E1 -12855.364,E2 -12855.364} C_VEL
LIN {X 0,Y 374.773,Z 441.476,A -85,B 0,C 180,E1 -12856.168,E2 -12856.168} C_VEL
LIN {X 0,Y 374.044,Z 453.069,A -85,B 0,C 180,E1 -12857.247,E2 -12857.247} C_VEL
LIN {X 0,Y 373.075,Z 464.308,A -85,B 0,C 180,E1 -12858.584,E2 -12858.584} C_VEL
LIN {X 0,Y 372.223,Z 473.479,A -85,B 0,C 180,E1 -12859.943,E2 -12859.943} C_VEL
LIN {X 0,Y 371.439,Z 482.213,A -85,B 0,C 180,E1 -12861.569,E2 -12861.569} C_VEL
LIN {X 0,Y 370.631,Z 489.269,A -85,B 0,C 180,E1 -12863.195,E2 -12863.195} C_VEL
LIN {X 0,Y 369.999,Z 495.72,A -85,B 0,C 180,E1 -12865.098,E2 -12865.098} C_VEL
LIN {X 0,Y 369.563,Z 499.963,A -85,B 0,C 180,E1 -12866.731,E2 -12866.731} C_VEL
LIN {X 0,Y 369.307,Z 502.202,A -85,B 0,C 180,E1 -12867.82,E2 -12867.82} C_VEL
LIN {X 0,Y 369.121,Z 504.029,A -85,B 0,C 180,E1 -12868.91,E2 -12868.91} C_VEL
LIN {X 0,Y 369.02,Z 505.417,A -85,B 0,C 180,E1 -12870.001,E2 -12870.001} C_VEL
LIN {X 0,Y 368.903,Z 507.007,A -85,B 0,C 180,E1 -12872.185,E2 -12872.185} C_VEL
LIN {X 0,Y 368.765,Z 507.265,A -85,B 0,C 180,E1 -12873.279,E2 -12873.279} C_VEL
LIN {X 0,Y 369.038,Z 506.496,A -85,B 0,C 180,E1 -12875.465,E2 -12875.465} C_VEL
LIN {X 0,Y 369.334,Z 505.533,A -85,B 0,C 180,E1 -12876.557,E2 -12876.557} C_VEL
LIN {X 0,Y 369.455,Z 504.205,A -85,B 0,C 180,E1 -12877.653,E2 -12877.653} C_VEL
LIN {X 0,Y 369.875,Z 501.383,A -85,B 0,C 180,E1 -12879.296,E2 -12879.296} C_VEL
LIN {X 0,Y 370.426,Z 497.534,A -85,B 0,C 180,E1 -12880.938,E2 -12880.938} C_VEL
LIN {X 0,Y 371.057,Z 492.542,A -85,B 0,C 180,E1 -12882.582,E2 -12882.582} C_VEL
LIN {X 0,Y 371.727,Z 486.248,A -85,B 0,C 180,E1 -12884.229,E2 -12884.229} C_VEL
LIN {X 0,Y 372.734,Z 478.081,A -85,B 0,C 180,E1 -12885.924,E2 -12885.924} C_VEL
LIN {X 0,Y 373.611,Z 470.28,A -85,B 0,C 180,E1 -12887.235,E2 -12887.235} C_VEL
LIN {X 0,Y 374.576,Z 460.281,A -85,B 0,C 180,E1 -12888.601,E2 -12888.601} C_VEL
LIN {X 0,Y 375.438,Z 449.133,A -85,B 0,C 180,E1 -12889.824,E2 -12889.824} C_VEL
LIN {X 0,Y 376.206,Z 437.802,A -85,B 0,C 180,E1 -12890.791,E2 -12890.791} C_VEL
LIN {X 0,Y 376.798,Z 425.79,A -85,B 0,C 180,E1 -12891.572,E2 -12891.572} C_VEL
LIN {X 0,Y 374.364,Z 417.695,A -85,B 0,C 180,E1 -12892.15,E2 -12892.15} C_VEL
LIN {X 0,Y 369.714,Z 405.593,A -85,B 0,C 180,E1 -12892.887,E2 -12892.887} C_VEL
LIN {X 0,Y 368.934,Z 403.154,A -85,B 0,C 180,E1 -12893.031,E2 -12893.031} C_VEL
LIN {X 0,Y 368.982,Z 403.149,A -85,B 0,C 180,E1 -12896.577,E2 -12896.577} C_VEL
LIN {X 0,Y 368.289,Z 403.236,A -85,B 0,C 180,E1 -12897.488,E2 -12897.488} C_VEL
LIN {X 0,Y 365.415,Z 403.598,A -85,B 0,C 180,E1 -12898.967,E2 -12898.967} C_VEL
LIN {X 0,Y 362.988,Z 403.902,A -85,B 0,C 180,E1 -12900.164,E2 -12900.164} C_VEL
LIN {X 0,Y 361.939,Z 404.03,A -85,B 0,C 180,E1 -12901.09,E2 -12901.09} C_VEL
LIN {X 0,Y 361.848,Z 404.04,A -85,B 0,C 180,E1 -12901.404,E2 -12901.404} C_VEL
LIN {X 0,Y 361.86,Z 404.039,A -85,B 0,C 180,E1 -12904.281,E2 -12904.281} C_VEL
LIN {X 0,Y 361.869,Z 404.027,A -85,B 0,C 180,E1 -12907.223,E2 -12907.223} C_VEL
LIN {X 0,Y 361.841,Z 404.04,A -85,B 0,C 180,E1 -12910.756,E2 -12910.756} C_VEL
LIN {X 0,Y 361.824,Z 404.041,A -85,B 0,C 180,E1 -12914.368,E2 -12914.368} C_VEL
LIN {X 0,Y 361.849,Z 404.035,A -85,B 0,C 180,E1 -12917.567,E2 -12917.567} C_VEL
LIN {X 0,Y 361.875,Z 404.004,A -85,B 0,C 180,E1 -12920.973,E2 -12920.973} C_VEL
LIN {X 0,Y 361.88,Z 404.032,A -85,B 0,C 180,E1 -12924.655,E2 -12924.655} C_VEL
LIN {X 0,Y 361.843,Z 404.018,A -85,B 0,C 180,E1 -12928.371,E2 -12928.371} C_VEL
LIN {X 0,Y 361.913,Z 404.007,A -85,B 0,C 180,E1 -12932.221,E2 -12932.221} C_VEL
LIN {X 0,Y 361.931,Z 404.023,A -85,B 0,C 180,E1 -12934.71,E2 -12934.71} C_VEL
LIN {X 0,Y 361.866,Z 404.034,A -85,B 0,C 180,E1 -12938.345,E2 -12938.345} C_VEL
LIN {X 0,Y 361.92,Z 404.029,A -85,B 0,C 180,E1 -12939.354,E2 -12939.354} C_VEL
LIN {X 0,Y 366.203,Z 418.485,A -85,B 0,C 180,E1 -12940.567,E2 -12940.567} C_VEL
LIN {X 0,Y 368.533,Z 426.783,A -85,B 0,C 180,E1 -12941.371,E2 -12941.371} C_VEL
LIN {X 0,Y 367.493,Z 440.09,A -85,B 0,C 180,E1 -12942.656,E2 -12942.656} C_VEL
LIN {X 0,Y 366.424,Z 452.795,A -85,B 0,C 180,E1 -12944.165,E2 -12944.165} C_VEL
LIN {X 0,Y 365.308,Z 464.155,A -85,B 0,C 180,E1 -12945.801,E2 -12945.801} C_VEL
LIN {X 0,Y 364.437,Z 473.701,A -85,B 0,C 180,E1 -12947.47,E2 -12947.47} C_VEL
LIN {X 0,Y 363.592,Z 482.879,A -85,B 0,C 180,E1 -12949.418,E2 -12949.418} C_VEL
LIN {X 0,Y 363.019,Z 489.409,A -85,B 0,C 180,E1 -12951.09,E2 -12951.09} C_VEL
LIN {X 0,Y 362.541,Z 496.402,A -85,B 0,C 180,E1 -12953.32,E2 -12953.32} C_VEL
LIN {X 0,Y 361.958,Z 501.785,A -85,B 0,C 180,E1 -12955.545,E2 -12955.545} C_VEL
LIN {X 0,Y 361.905,Z 505.604,A -85,B 0,C 180,E1 -12957.774,E2 -12957.774} C_VEL
LIN {X 0,Y 361.952,Z 507.991,A -85,B 0,C 180,E1 -12960,E2 -12960} C_VEL
LIN {X 0,Y 362.147,Z 509.032,A -85,B 0,C 180,E1 -12962.224,E2 -12962.224} C_VEL
LIN {X 0,Y 362.421,Z 508.755,A -85,B 0,C 180,E1 -12964.448,E2 -12964.448} C_VEL
LIN {X 0,Y 362.91,Z 507.146,A -85,B 0,C 180,E1 -12966.672,E2 -12966.672} C_VEL
LIN {X 0,Y 363.754,Z 504.14,A -85,B 0,C 180,E1 -12968.891,E2 -12968.891} C_VEL
LIN {X 0,Y 364.532,Z 501.004,A -85,B 0,C 180,E1 -12970.497,E2 -12970.497} C_VEL
LIN {X 0,Y 365.72,Z 495.252,A -85,B 0,C 180,E1 -12972.767,E2 -12972.767} C_VEL
LIN {X 0,Y 367.072,Z 488.865,A -85,B 0,C 180,E1 -12974.696,E2 -12974.696} C_VEL
LIN {X 0,Y 368.693,Z 480.877,A -85,B 0,C 180,E1 -12976.614,E2 -12976.614} C_VEL
LIN {X 0,Y 370.314,Z 472.425,A -85,B 0,C 180,E1 -12978.277,E2 -12978.277} C_VEL
LIN {X 0,Y 371.997,Z 462.613,A -85,B 0,C 180,E1 -12979.881,E2 -12979.881} C_VEL
LIN {X 0,Y 373.789,Z 451.585,A -85,B 0,C 180,E1 -12981.364,E2 -12981.364} C_VEL
LIN {X 0,Y 375.555,Z 439.315,A -85,B 0,C 180,E1 -12982.718,E2 -12982.718} C_VEL
LIN {X 0,Y 375.773,Z 435.42,A -85,B 0,C 180,E1 -12983.126,E2 -12983.126} C_VEL
LIN {X 0,Y 372.177,Z 424.679,A -85,B 0,C 180,E1 -12984.682,E2 -12984.682} C_VEL
LIN {X 0,Y 367.881,Z 415.251,A -85,B 0,C 180,E1 -12986.117,E2 -12986.117} C_VEL
LIN {X 0,Y 363.821,Z 408.033,A -85,B 0,C 180,E1 -12987.302,E2 -12987.302} C_VEL
LIN {X 0,Y 362.26,Z 405.496,A -85,B 0,C 180,E1 -12987.75,E2 -12987.75} C_VEL
LIN {X 0,Y 361.904,Z 404.031,A -85,B 0,C 180,E1 -12987.936,E2 -12987.936} C_VEL
LIN {X 0,Y 361.841,Z 404.037,A -85,B 0,C 180,E1 -12991.629,E2 -12991.629} C_VEL
LIN {X 0,Y 361.907,Z 404.154,A -85,B 0,C 180,E1 -12995.351,E2 -12995.351} C_VEL
LIN {X 0,Y 362.464,Z 406.824,A -85,B 0,C 180,E1 -12998.35,E2 -12998.35} C_VEL
LIN {X 0,Y 363.141,Z 410.039,A -85,B 0,C 180,E1 -13001.148,E2 -13001.148} C_VEL
LIN {X 0,Y 364.213,Z 414.749,A -85,B 0,C 180,E1 -13004.44,E2 -13004.44} C_VEL
LIN {X 0,Y 365.309,Z 420.483,A -85,B 0,C 180,E1 -13007.673,E2 -13007.673} C_VEL
LIN {X 0,Y 365.96,Z 424.859,A -85,B 0,C 180,E1 -13009.795,E2 -13009.795} C_VEL
LIN {X 0,Y 365.061,Z 430.234,A -85,B 0,C 180,E1 -13011.971,E2 -13011.971} C_VEL
LIN {X 0,Y 363.637,Z 441.698,A -85,B 0,C 180,E1 -13016.207,E2 -13016.207} C_VEL
LIN {X 0,Y 362.792,Z 452.166,A -85,B 0,C 180,E1 -13019.756,E2 -13019.756} C_VEL
LIN {X 0,Y 362.208,Z 461.339,A -85,B 0,C 180,E1 -13022.694,E2 -13022.694} C_VEL
LIN {X 0,Y 363.151,Z 465.675,A -85,B 0,C 180,E1 -13023.037,E2 -13023.037} C_VEL
LIN {X 0,Y 363.933,Z 468.615,A -85,B 0,C 180,E1 -13023.292,E2 -13023.292} C_VEL
LIN {X 0,Y 366.623,Z 480.773,A -85,B 0,C 180,E1 -13024.285,E2 -13024.285} C_VEL
LIN {X 0,Y 368.659,Z 495.702,A -85,B 0,C 180,E1 -13025.474,E2 -13025.474} C_VEL
LIN {X 0,Y 369.22,Z 507.659,A -85,B 0,C 180,E1 -13026.438,E2 -13026.438} C_VEL
LIN {X 0,Y 368.773,Z 522.746,A -85,B 0,C 180,E1 -13027.741,E2 -13027.741} C_VEL
LIN {X 0,Y 368.326,Z 534.312,A -85,B 0,C 180,E1 -13028.904,E2 -13028.904} C_VEL
LIN {X 0,Y 366.287,Z 547.691,A -85,B 0,C 180,E1 -13030.386,E2 -13030.386} C_VEL
LIN {X 0,Y 364.587,Z 559.995,A -85,B 0,C 180,E1 -13032.035,E2 -13032.035} C_VEL
LIN {X 0,Y 363.218,Z 570.482,A -85,B 0,C 180,E1 -13033.705,E2 -13033.705} C_VEL
LIN {X 0,Y 362.133,Z 580.835,A -85,B 0,C 180,E1 -13035.677,E2 -13035.677} C_VEL
LIN {X 0,Y 361.397,Z 589.4,A -85,B 0,C 180,E1 -13037.647,E2 -13037.647} C_VEL
LIN {X 0,Y 361.109,Z 595.522,A -85,B 0,C 180,E1 -13039.344,E2 -13039.344} C_VEL
LIN {X 0,Y 361.007,Z 602.175,A -85,B 0,C 180,E1 -13041.603,E2 -13041.603} C_VEL
LIN {X 0,Y 361.153,Z 607.165,A -85,B 0,C 180,E1 -13043.855,E2 -13043.855} C_VEL
LIN {X 0,Y 361.404,Z 609.842,A -85,B 0,C 180,E1 -13045.538,E2 -13045.538} C_VEL
LIN {X 0,Y 361.444,Z 612.086,A -85,B 0,C 180,E1 -13047.77,E2 -13047.77} C_VEL
LIN {X 0,Y 361.649,Z 612.67,A -85,B 0,C 180,E1 -13048.885,E2 -13048.885} C_VEL
LIN {X 0,Y 361.811,Z 612.87,A -85,B 0,C 180,E1 -13049.999,E2 -13049.999} C_VEL
LIN {X 0,Y 361.457,Z 612.031,A -85,B 0,C 180,E1 -13052.227,E2 -13052.227} C_VEL
LIN {X 0,Y 361.405,Z 611.055,A -85,B 0,C 180,E1 -13053.343,E2 -13053.343} C_VEL
LIN {X 0,Y 361.372,Z 609.684,A -85,B 0,C 180,E1 -13054.46,E2 -13054.46} C_VEL
LIN {X 0,Y 361.237,Z 606.857,A -85,B 0,C 180,E1 -13056.141,E2 -13056.141} C_VEL
LIN {X 0,Y 361.109,Z 601.643,A -85,B 0,C 180,E1 -13058.392,E2 -13058.392} C_VEL
LIN {X 0,Y 361.172,Z 596.504,A -85,B 0,C 180,E1 -13060.085,E2 -13060.085} C_VEL
LIN {X 0,Y 361.461,Z 589.108,A -85,B 0,C 180,E1 -13062.063,E2 -13062.063} C_VEL
LIN {X 0,Y 361.955,Z 580.773,A -85,B 0,C 180,E1 -13063.871,E2 -13063.871} C_VEL
LIN {X 0,Y 362.727,Z 572.025,A -85,B 0,C 180,E1 -13065.449,E2 -13065.449} C_VEL
LIN {X 0,Y 363.808,Z 560.735,A -85,B 0,C 180,E1 -13067.132,E2 -13067.132} C_VEL
LIN {X 0,Y 364.947,Z 549.386,A -85,B 0,C 180,E1 -13068.525,E2 -13068.525} C_VEL
LIN {X 0,Y 366.076,Z 538.409,A -85,B 0,C 180,E1 -13069.644,E2 -13069.644} C_VEL
LIN {X 0,Y 366.832,Z 528.964,A -85,B 0,C 180,E1 -13070.464,E2 -13070.464} C_VEL
LIN {X 0,Y 365.825,Z 515.51,A -85,B 0,C 180,E1 -13071.483,E2 -13071.483} C_VEL
LIN {X 0,Y 364.237,Z 500.307,A -85,B 0,C 180,E1 -13072.4,E2 -13072.4} C_VEL
LIN {X 0,Y 362.419,Z 484.681,A -85,B 0,C 180,E1 -13073.11,E2 -13073.11} C_VEL
LIN {X 0,Y 361.963,Z 480.357,A -85,B 0,C 180,E1 -13073.302,E2 -13073.302} C_VEL
LIN {X 0,Y 362.767,Z 467.96,A -85,B 0,C 180,E1 -13077.274,E2 -13077.274} C_VEL
LIN {X 0,Y 363.897,Z 455.213,A -85,B 0,C 180,E1 -13081.428,E2 -13081.428} C_VEL
LIN {X 0,Y 365.066,Z 443.612,A -85,B 0,C 180,E1 -13085.276,E2 -13085.276} C_VEL
LIN {X 0,Y 366.421,Z 431.9,A -85,B 0,C 180,E1 -13089.266,E2 -13089.266} C_VEL
LIN {X 0,Y 366.563,Z 427.867,A -85,B 0,C 180,E1 -13090.681,E2 -13090.681} C_VEL
LIN {X 0,Y 365.427,Z 421.584,A -85,B 0,C 180,E1 -13093.044,E2 -13093.044} C_VEL
LIN {X 0,Y 363.552,Z 412.363,A -85,B 0,C 180,E1 -13096.666,E2 -13096.666} C_VEL
LIN {X 0,Y 361.894,Z 404.034,A -85,B 0,C 180,E1 -13100.144,E2 -13100.144} C_VEL
LIN {X 0,Y 361.861,Z 404.036,A -85,B 0,C 180,E1 -13102.981,E2 -13102.981} C_VEL
LIN {X 0,Y 361.849,Z 404.034,A -85,B 0,C 180,E1 -13106.63,E2 -13106.63} C_VEL
LIN {X 0,Y 361.867,Z 404.032,A -85,B 0,C 180,E1 -13109.672,E2 -13109.672} C_VEL
LIN {X 0,Y 361.945,Z 404.024,A -85,B 0,C 180,E1 -13113.475,E2 -13113.475} C_VEL
LIN {X 0,Y 361.88,Z 404.035,A -85,B 0,C 180,E1 -13117.144,E2 -13117.144} C_VEL
LIN {X 0,Y 361.896,Z 404.03,A -85,B 0,C 180,E1 -13120.723,E2 -13120.723} C_VEL
LIN {X 0,Y 361.922,Z 404.03,A -85,B 0,C 180,E1 -13123.066,E2 -13123.066} C_VEL
LIN {X 0,Y 361.989,Z 404.017,A -85,B 0,C 180,E1 -13126.528,E2 -13126.528} C_VEL
LIN {X 0,Y 362.026,Z 404.011,A -85,B 0,C 180,E1 -13129.938,E2 -13129.938} C_VEL
LIN {X 0,Y 362.14,Z 403.997,A -85,B 0,C 180,E1 -13132.193,E2 -13132.193} C_VEL
LIN {X 0,Y 362.108,Z 404.002,A -85,B 0,C 180,E1 -13134.431,E2 -13134.431} C_VEL
LIN {X 0,Y 362.273,Z 403.98,A -85,B 0,C 180,E1 -13137.777,E2 -13137.777} C_VEL
LIN {X 0,Y 362.419,Z 403.962,A -85,B 0,C 180,E1 -13140,E2 -13140} C_VEL
LIN {X 0,Y 362.273,Z 403.981,A -85,B 0,C 180,E1 -13142.224,E2 -13142.224} C_VEL
LIN {X 0,Y 362.162,Z 403.999,A -85,B 0,C 180,E1 -13146.687,E2 -13146.687} C_VEL
LIN {X 0,Y 362.066,Z 404.011,A -85,B 0,C 180,E1 -13148.934,E2 -13148.934} C_VEL
LIN {X 0,Y 361.958,Z 404.021,A -85,B 0,C 180,E1 -13152.333,E2 -13152.333} C_VEL
LIN {X 0,Y 361.953,Z 404.025,A -85,B 0,C 180,E1 -13154.621,E2 -13154.621} C_VEL
LIN {X 0,Y 361.95,Z 404.021,A -85,B 0,C 180,E1 -13158.1,E2 -13158.1} C_VEL
LIN {X 0,Y 361.883,Z 404.029,A -85,B 0,C 180,E1 -13161.654,E2 -13161.654} C_VEL
LIN {X 0,Y 361.92,Z 404.025,A -85,B 0,C 180,E1 -13165.291,E2 -13165.291} C_VEL
LIN {X 0,Y 361.91,Z 404.025,A -85,B 0,C 180,E1 -13167.779,E2 -13167.779} C_VEL
LIN {X 0,Y 361.839,Z 404.035,A -85,B 0,C 180,E1 -13171.286,E2 -13171.286} C_VEL
LIN {X 0,Y 361.847,Z 404.036,A -85,B 0,C 180,E1 -13174.282,E2 -13174.282} C_VEL
LIN {X 0,Y 361.858,Z 404.032,A -85,B 0,C 180,E1 -13177.225,E2 -13177.225} C_VEL
LIN {X 0,Y 361.831,Z 404.039,A -85,B 0,C 180,E1 -13180.757,E2 -13180.757} C_VEL
LIN {X 0,Y 361.842,Z 404.038,A -85,B 0,C 180,E1 -13184.365,E2 -13184.365} C_VEL
LIN {X 0,Y 361.852,Z 404.032,A -85,B 0,C 180,E1 -13187.566,E2 -13187.566} C_VEL
LIN {X 0,Y 361.871,Z 404.032,A -85,B 0,C 180,E1 -13190.974,E2 -13190.974} C_VEL
LIN {X 0,Y 361.872,Z 404.034,A -85,B 0,C 180,E1 -13194.657,E2 -13194.657} C_VEL
LIN {X 0,Y 361.836,Z 404.041,A -85,B 0,C 180,E1 -13198.372,E2 -13198.372} C_VEL
LIN {X 0,Y 361.907,Z 404.03,A -85,B 0,C 180,E1 -13202.223,E2 -13202.223} C_VEL
LIN {X 0,Y 361.928,Z 404.026,A -85,B 0,C 180,E1 -13204.712,E2 -13204.712} C_VEL
LIN {X 0,Y 361.892,Z 404.034,A -85,B 0,C 180,E1 -13208.349,E2 -13208.349} C_VEL
LIN {X 0,Y 361.968,Z 404.022,A -85,B 0,C 180,E1 -13212.063,E2 -13212.063} C_VEL
LIN {X 0,Y 361.924,Z 404.141,A -85,B 0,C 180,E1 -13213.444,E2 -13213.444} C_VEL
LIN {X 0,Y 366.353,Z 416.846,A -85,B 0,C 180,E1 -13214.131,E2 -13214.131} C_VEL
LIN {X 0,Y 368.649,Z 424.091,A -85,B 0,C 180,E1 -13214.613,E2 -13214.613} C_VEL
LIN {X 0,Y 368.368,Z 435.825,A -85,B 0,C 180,E1 -13215.358,E2 -13215.358} C_VEL
LIN {X 0,Y 367.722,Z 447.521,A -85,B 0,C 180,E1 -13216.32,E2 -13216.32} C_VEL
LIN {X 0,Y 366.939,Z 458.059,A -85,B 0,C 180,E1 -13217.418,E2 -13217.418} C_VEL
LIN {X 0,Y 366.027,Z 468.065,A -85,B 0,C 180,E1 -13218.722,E2 -13218.722} C_VEL
LIN {X 0,Y 364.994,Z 477.811,A -85,B 0,C 180,E1 -13220.302,E2 -13220.302} C_VEL
LIN {X 0,Y 364.176,Z 485.906,A -85,B 0,C 180,E1 -13221.958,E2 -13221.958} C_VEL
LIN {X 0,Y 363.476,Z 491.457,A -85,B 0,C 180,E1 -13223.339,E2 -13223.339} C_VEL
LIN {X 0,Y 363.01,Z 496.821,A -85,B 0,C 180,E1 -13225.003,E2 -13225.003} C_VEL
LIN {X 0,Y 362.559,Z 501.041,A -85,B 0,C 180,E1 -13226.667,E2 -13226.667} C_VEL
LIN {X 0,Y 362.291,Z 503.271,A -85,B 0,C 180,E1 -13227.778,E2 -13227.778} C_VEL
LIN {X 0,Y 362.1,Z 505.087,A -85,B 0,C 180,E1 -13228.889,E2 -13228.889} C_VEL
LIN {X 0,Y 361.999,Z 506.454,A -85,B 0,C 180,E1 -13230.001,E2 -13230.001} C_VEL
LIN {X 0,Y 361.878,Z 508.026,A -85,B 0,C 180,E1 -13232.227,E2 -13232.227} C_VEL
LIN {X 0,Y 361.741,Z 508.271,A -85,B 0,C 180,E1 -13233.343,E2 -13233.343} C_VEL
LIN {X 0,Y 362.036,Z 507.475,A -85,B 0,C 180,E1 -13235.571,E2 -13235.571} C_VEL
LIN {X 0,Y 362.345,Z 506.503,A -85,B 0,C 180,E1 -13236.684,E2 -13236.684} C_VEL
LIN {X 0,Y 362.481,Z 505.155,A -85,B 0,C 180,E1 -13237.801,E2 -13237.801} C_VEL
LIN {X 0,Y 362.937,Z 502.312,A -85,B 0,C 180,E1 -13239.475,E2 -13239.475} C_VEL
LIN {X 0,Y 363.516,Z 498.438,A -85,B 0,C 180,E1 -13241.149,E2 -13241.149} C_VEL
LIN {X 0,Y 364.165,Z 493.422,A -85,B 0,C 180,E1 -13242.824,E2 -13242.824} C_VEL
LIN {X 0,Y 365.056,Z 485.912,A -85,B 0,C 180,E1 -13244.78,E2 -13244.78} C_VEL
LIN {X 0,Y 365.921,Z 479.075,A -85,B 0,C 180,E1 -13246.194,E2 -13246.194} C_VEL
LIN {X 0,Y 366.884,Z 471.051,A -85,B 0,C 180,E1 -13247.561,E2 -13247.561} C_VEL
LIN {X 0,Y 367.9,Z 460.986,A -85,B 0,C 180,E1 -13248.952,E2 -13248.952} C_VEL
LIN {X 0,Y 368.79,Z 449.811,A -85,B 0,C 180,E1 -13250.192,E2 -13250.192} C_VEL
LIN {X 0,Y 369.599,Z 438.301,A -85,B 0,C 180,E1 -13251.18,E2 -13251.18} C_VEL
LIN {X 0,Y 370.117,Z 426.779,A -85,B 0,C 180,E1 -13251.943,E2 -13251.943} C_VEL
LIN {X 0,Y 366.002,Z 414.663,A -85,B 0,C 180,E1 -13252.823,E2 -13252.823} C_VEL
LIN {X 0,Y 362.01,Z 404.525,A -85,B 0,C 180,E1 -13253.418,E2 -13253.418} C_VEL
LIN {X 0,Y 361.919,Z 404.027,A -85,B 0,C 180,E1 -13253.461,E2 -13253.461} C_VEL
LIN {X 0,Y 361.949,Z 404.025,A -85,B 0,C 180,E1 -13256.722,E2 -13256.722} C_VEL
LIN {X 0,Y 361.881,Z 404.035,A -85,B 0,C 180,E1 -13260.328,E2 -13260.328} C_VEL
LIN {X 0,Y 361.848,Z 404.04,A -85,B 0,C 180,E1 -13261.404,E2 -13261.404} C_VEL
LIN {X 0,Y 361.168,Z 404.125,A -85,B 0,C 180,E1 -13262.332,E2 -13262.332} C_VEL
LIN {X 0,Y 358.316,Z 404.479,A -85,B 0,C 180,E1 -13263.841,E2 -13263.841} C_VEL
LIN {X 0,Y 355.913,Z 404.779,A -85,B 0,C 180,E1 -13265.063,E2 -13265.063} C_VEL
LIN {X 0,Y 354.885,Z 404.906,A -85,B 0,C 180,E1 -13266.007,E2 -13266.007} C_VEL
LIN {X 0,Y 354.803,Z 404.915,A -85,B 0,C 180,E1 -13266.327,E2 -13266.327} C_VEL
LIN {X 0,Y 354.83,Z 404.906,A -85,B 0,C 180,E1 -13269.424,E2 -13269.424} C_VEL
LIN {X 0,Y 354.794,Z 404.914,A -85,B 0,C 180,E1 -13272.867,E2 -13272.867} C_VEL
LIN {X 0,Y 354.781,Z 404.913,A -85,B 0,C 180,E1 -13276.105,E2 -13276.105} C_VEL
LIN {X 0,Y 354.797,Z 404.907,A -85,B 0,C 180,E1 -13279.18,E2 -13279.18} C_VEL
LIN {X 0,Y 354.813,Z 404.891,A -85,B 0,C 180,E1 -13282.402,E2 -13282.402} C_VEL
LIN {X 0,Y 354.818,Z 404.911,A -85,B 0,C 180,E1 -13284.941,E2 -13284.941} C_VEL
LIN {X 0,Y 354.798,Z 404.895,A -85,B 0,C 180,E1 -13288.405,E2 -13288.405} C_VEL
LIN {X 0,Y 354.851,Z 404.876,A -85,B 0,C 180,E1 -13291.619,E2 -13291.619} C_VEL
LIN {X 0,Y 354.903,Z 404.901,A -85,B 0,C 180,E1 -13294.172,E2 -13294.172} C_VEL
LIN {X 0,Y 354.82,Z 404.914,A -85,B 0,C 180,E1 -13297.893,E2 -13297.893} C_VEL
LIN {X 0,Y 354.9,Z 405.093,A -85,B 0,C 180,E1 -13299.068,E2 -13299.068} C_VEL
LIN {X 0,Y 359.224,Z 419.519,A -85,B 0,C 180,E1 -13300.313,E2 -13300.313} C_VEL
LIN {X 0,Y 361.575,Z 427.92,A -85,B 0,C 180,E1 -13301.147,E2 -13301.147} C_VEL
LIN {X 0,Y 360.608,Z 440.8,A -85,B 0,C 180,E1 -13302.417,E2 -13302.417} C_VEL
LIN {X 0,Y 359.555,Z 452.964,A -85,B 0,C 180,E1 -13303.877,E2 -13303.877} C_VEL
LIN {X 0,Y 358.391,Z 464.327,A -85,B 0,C 180,E1 -13305.521,E2 -13305.521} C_VEL
LIN {X 0,Y 357.507,Z 474.054,A -85,B 0,C 180,E1 -13307.223,E2 -13307.223} C_VEL
LIN {X 0,Y 356.743,Z 482.183,A -85,B 0,C 180,E1 -13308.926,E2 -13308.926} C_VEL
LIN {X 0,Y 356.048,Z 490.024,A -85,B 0,C 180,E1 -13310.914,E2 -13310.914} C_VEL
LIN {X 0,Y 355.538,Z 497.133,A -85,B 0,C 180,E1 -13313.188,E2 -13313.188} C_VEL
LIN {X 0,Y 355.191,Z 501.389,A -85,B 0,C 180,E1 -13314.891,E2 -13314.891} C_VEL
LIN {X 0,Y 354.786,Z 504.779,A -85,B 0,C 180,E1 -13316.593,E2 -13316.593} C_VEL
LIN {X 0,Y 354.913,Z 507.968,A -85,B 0,C 180,E1 -13318.865,E2 -13318.865} C_VEL
LIN {X 0,Y 355.001,Z 509.785,A -85,B 0,C 180,E1 -13321.134,E2 -13321.134} C_VEL
LIN {X 0,Y 355.299,Z 510.252,A -85,B 0,C 180,E1 -13323.402,E2 -13323.402} C_VEL
LIN {X 0,Y 355.692,Z 509.407,A -85,B 0,C 180,E1 -13325.669,E2 -13325.669} C_VEL
LIN {X 0,Y 356.419,Z 507.193,A -85,B 0,C 180,E1 -13327.934,E2 -13327.934} C_VEL
LIN {X 0,Y 357.473,Z 503.579,A -85,B 0,C 180,E1 -13330.191,E2 -13330.191} C_VEL
LIN {X 0,Y 358.652,Z 498.474,A -85,B 0,C 180,E1 -13332.448,E2 -13332.448} C_VEL
LIN {X 0,Y 359.805,Z 493.538,A -85,B 0,C 180,E1 -13334.132,E2 -13334.132} C_VEL
LIN {X 0,Y 361.408,Z 486.446,A -85,B 0,C 180,E1 -13336.087,E2 -13336.087} C_VEL
LIN {X 0,Y 363.285,Z 477.633,A -85,B 0,C 180,E1 -13338.031,E2 -13338.031} C_VEL
LIN {X 0,Y 365.073,Z 468.493,A -85,B 0,C 180,E1 -13339.687,E2 -13339.687} C_VEL
LIN {X 0,Y 367.056,Z 457.511,A -85,B 0,C 180,E1 -13341.333,E2 -13341.333} C_VEL
LIN {X 0,Y 368.982,Z 445.741,A -85,B 0,C 180,E1 -13342.768,E2 -13342.768} C_VEL
LIN {X 0,Y 369.911,Z 438.68,A -85,B 0,C 180,E1 -13343.514,E2 -13343.514} C_VEL
LIN {X 0,Y 367.109,Z 429.556,A -85,B 0,C 180,E1 -13344.908,E2 -13344.908} C_VEL
LIN {X 0,Y 363.78,Z 421.622,A -85,B 0,C 180,E1 -13346.19,E2 -13346.19} C_VEL
LIN {X 0,Y 360.227,Z 414.676,A -85,B 0,C 180,E1 -13347.38,E2 -13347.38} C_VEL
LIN {X 0,Y 357.042,Z 409.176,A -85,B 0,C 180,E1 -13348.393,E2 -13348.393} C_VEL
LIN {X 0,Y 355.278,Z 406.528,A -85,B 0,C 180,E1 -13348.932,E2 -13348.932} C_VEL
LIN {X 0,Y 354.875,Z 404.905,A -85,B 0,C 180,E1 -13349.142,E2 -13349.142} C_VEL
LIN {X 0,Y 354.822,Z 404.961,A -85,B 0,C 180,E1 -13353.343,E2 -13353.343} C_VEL
LIN {X 0,Y 355.313,Z 407.19,A -85,B 0,C 180,E1 -13356.398,E2 -13356.398} C_VEL
LIN {X 0,Y 356.01,Z 410.398,A -85,B 0,C 180,E1 -13359.654,E2 -13359.654} C_VEL
LIN {X 0,Y 356.99,Z 415.034,A -85,B 0,C 180,E1 -13363.245,E2 -13363.245} C_VEL
LIN {X 0,Y 358.124,Z 420.404,A -85,B 0,C 180,E1 -13366.561,E2 -13366.561} C_VEL
LIN {X 0,Y 358.95,Z 425.087,A -85,B 0,C 180,E1 -13369.011,E2 -13369.011} C_VEL
LIN {X 0,Y 359.081,Z 426.694,A -85,B 0,C 180,E1 -13369.767,E2 -13369.767} C_VEL
LIN {X 0,Y 357.847,Z 433.367,A -85,B 0,C 180,E1 -13372.494,E2 -13372.494} C_VEL
LIN {X 0,Y 356.554,Z 444.037,A -85,B 0,C 180,E1 -13376.501,E2 -13376.501} C_VEL
LIN {X 0,Y 355.623,Z 455.376,A -85,B 0,C 180,E1 -13380.406,E2 -13380.406} C_VEL
LIN {X 0,Y 355.357,Z 459.126,A -85,B 0,C 180,E1 -13381.602,E2 -13381.602} C_VEL
LIN {X 0,Y 356.466,Z 463.827,A -85,B 0,C 180,E1 -13382.026,E2 -13382.026} C_VEL
LIN {X 0,Y 358.565,Z 472.12,A -85,B 0,C 180,E1 -13382.794,E2 -13382.794} C_VEL
LIN {X 0,Y 360.901,Z 484.026,A -85,B 0,C 180,E1 -13383.847,E2 -13383.847} C_VEL
LIN {X 0,Y 362.54,Z 498.213,A -85,B 0,C 180,E1 -13385.062,E2 -13385.062} C_VEL
LIN {X 0,Y 362.86,Z 511.171,A -85,B 0,C 180,E1 -13386.184,E2 -13386.184} C_VEL
LIN {X 0,Y 362.062,Z 526.396,A -85,B 0,C 180,E1 -13387.607,E2 -13387.607} C_VEL
LIN {X 0,Y 361.484,Z 536.016,A -85,B 0,C 180,E1 -13388.65,E2 -13388.65} C_VEL
LIN {X 0,Y 359.17,Z 550.024,A -85,B 0,C 180,E1 -13390.305,E2 -13390.305} C_VEL
LIN {X 0,Y 357.514,Z 561.559,A -85,B 0,C 180,E1 -13391.963,E2 -13391.963} C_VEL
LIN {X 0,Y 356.132,Z 571.586,A -85,B 0,C 180,E1 -13393.666,E2 -13393.666} C_VEL
LIN {X 0,Y 355.022,Z 581.461,A -85,B 0,C 180,E1 -13395.673,E2 -13395.673} C_VEL
LIN {X 0,Y 354.29,Z 589.684,A -85,B 0,C 180,E1 -13397.686,E2 -13397.686} C_VEL
LIN {X 0,Y 353.997,Z 596.472,A -85,B 0,C 180,E1 -13399.706,E2 -13399.706} C_VEL
LIN {X 0,Y 353.943,Z 602.603,A -85,B 0,C 180,E1 -13402.009,E2 -13402.009} C_VEL
LIN {X 0,Y 354.086,Z 606.166,A -85,B 0,C 180,E1 -13403.732,E2 -13403.732} C_VEL
LIN {X 0,Y 354.326,Z 608.822,A -85,B 0,C 180,E1 -13405.448,E2 -13405.448} C_VEL
LIN {X 0,Y 354.41,Z 611.027,A -85,B 0,C 180,E1 -13407.726,E2 -13407.726} C_VEL
LIN {X 0,Y 354.626,Z 611.589,A -85,B 0,C 180,E1 -13408.863,E2 -13408.863} C_VEL
LIN {X 0,Y 354.802,Z 611.768,A -85,B 0,C 180,E1 -13409.999,E2 -13409.999} C_VEL
LIN {X 0,Y 354.44,Z 610.857,A -85,B 0,C 180,E1 -13412.272,E2 -13412.272} C_VEL
LIN {X 0,Y 354.384,Z 609.841,A -85,B 0,C 180,E1 -13413.41,E2 -13413.41} C_VEL
LIN {X 0,Y 354.343,Z 608.436,A -85,B 0,C 180,E1 -13414.549,E2 -13414.549} C_VEL
LIN {X 0,Y 354.193,Z 605.576,A -85,B 0,C 180,E1 -13416.264,E2 -13416.264} C_VEL
LIN {X 0,Y 354.087,Z 601.723,A -85,B 0,C 180,E1 -13417.985,E2 -13417.985} C_VEL
LIN {X 0,Y 354.106,Z 596.883,A -85,B 0,C 180,E1 -13419.711,E2 -13419.711} C_VEL
LIN {X 0,Y 354.343,Z 589.826,A -85,B 0,C 180,E1 -13421.728,E2 -13421.728} C_VEL
LIN {X 0,Y 354.833,Z 581.046,A -85,B 0,C 180,E1 -13423.748,E2 -13423.748} C_VEL
LIN {X 0,Y 355.647,Z 571.906,A -85,B 0,C 180,E1 -13425.471,E2 -13425.471} C_VEL
LIN {X 0,Y 356.701,Z 560.86,A -85,B 0,C 180,E1 -13427.189,E2 -13427.189} C_VEL
LIN {X 0,Y 357.878,Z 549.751,A -85,B 0,C 180,E1 -13428.608,E2 -13428.608} C_VEL
LIN {X 0,Y 359.058,Z 538.381,A -85,B 0,C 180,E1 -13429.814,E2 -13429.814} C_VEL
LIN {X 0,Y 359.83,Z 529.836,A -85,B 0,C 180,E1 -13430.582,E2 -13430.582} C_VEL
LIN {X 0,Y 358.804,Z 515.83,A -85,B 0,C 180,E1 -13431.696,E2 -13431.696} C_VEL
LIN {X 0,Y 357.242,Z 500.52,A -85,B 0,C 180,E1 -13432.665,E2 -13432.665} C_VEL
LIN {X 0,Y 355.463,Z 484.537,A -85,B 0,C 180,E1 -13433.424,E2 -13433.424} C_VEL
LIN {X 0,Y 354.947,Z 479.531,A -85,B 0,C 180,E1 -13433.636,E2 -13433.636} C_VEL
LIN {X 0,Y 355.797,Z 467.176,A -85,B 0,C 180,E1 -13437.7,E2 -13437.7} C_VEL
LIN {X 0,Y 356.82,Z 455.876,A -85,B 0,C 180,E1 -13441.461,E2 -13441.461} C_VEL
LIN {X 0,Y 358.034,Z 444.332,A -85,B 0,C 180,E1 -13445.383,E2 -13445.383} C_VEL
LIN {X 0,Y 359.44,Z 432.606,A -85,B 0,C 180,E1 -13449.452,E2 -13449.452} C_VEL
LIN {X 0,Y 359.518,Z 428.47,A -85,B 0,C 180,E1 -13450.949,E2 -13450.949} C_VEL
LIN {X 0,Y 358.237,Z 421.946,A -85,B 0,C 180,E1 -13453.458,E2 -13453.458} C_VEL
LIN {X 0,Y 356.564,Z 413.555,A -85,B 0,C 180,E1 -13456.824,E2 -13456.824} C_VEL
LIN {X 0,Y 354.849,Z 404.91,A -85,B 0,C 180,E1 -13460.506,E2 -13460.506} C_VEL
LIN {X 0,Y 354.813,Z 404.91,A -85,B 0,C 180,E1 -13464.3,E2 -13464.3} C_VEL
LIN {X 0,Y 354.778,Z 404.915,A -85,B 0,C 180,E1 -13467.666,E2 -13467.666} C_VEL
LIN {X 0,Y 354.859,Z 404.905,A -85,B 0,C 180,E1 -13470.621,E2 -13470.621} C_VEL
LIN {X 0,Y 354.889,Z 404.9,A -85,B 0,C 180,E1 -13474.172,E2 -13474.172} C_VEL
LIN {X 0,Y 354.824,Z 404.908,A -85,B 0,C 180,E1 -13477.894,E2 -13477.894} C_VEL
LIN {X 0,Y 354.912,Z 404.897,A -85,B 0,C 180,E1 -13481.891,E2 -13481.891} C_VEL
LIN {X 0,Y 354.932,Z 404.894,A -85,B 0,C 180,E1 -13485.981,E2 -13485.981} C_VEL
LIN {X 0,Y 354.972,Z 404.89,A -85,B 0,C 180,E1 -13489.736,E2 -13489.736} C_VEL
LIN {X 0,Y 355.103,Z 404.873,A -85,B 0,C 180,E1 -13492.037,E2 -13492.037} C_VEL
LIN {X 0,Y 355.083,Z 404.877,A -85,B 0,C 180,E1 -13494.321,E2 -13494.321} C_VEL
LIN {X 0,Y 355.236,Z 404.857,A -85,B 0,C 180,E1 -13497.733,E2 -13497.733} C_VEL
LIN {X 0,Y 355.389,Z 404.838,A -85,B 0,C 180,E1 -13500,E2 -13500} C_VEL
LIN {X 0,Y 355.236,Z 404.858,A -85,B 0,C 180,E1 -13502.268,E2 -13502.268} C_VEL
LIN {X 0,Y 355.128,Z 404.876,A -85,B 0,C 180,E1 -13506.82,E2 -13506.82} C_VEL
LIN {X 0,Y 355.007,Z 404.887,A -85,B 0,C 180,E1 -13509.113,E2 -13509.113} C_VEL
LIN {X 0,Y 354.917,Z 404.9,A -85,B 0,C 180,E1 -13512.581,E2 -13512.581} C_VEL
LIN {X 0,Y 354.88,Z 404.902,A -85,B 0,C 180,E1 -13516.097,E2 -13516.097} C_VEL
LIN {X 0,Y 354.897,Z 404.902,A -85,B 0,C 180,E1 -13518.473,E2 -13518.473} C_VEL
LIN {X 0,Y 354.826,Z 404.909,A -85,B 0,C 180,E1 -13522.107,E2 -13522.107} C_VEL
LIN {X 0,Y 354.891,Z 404.9,A -85,B 0,C 180,E1 -13525.828,E2 -13525.828} C_VEL
LIN {X 0,Y 354.846,Z 404.904,A -85,B 0,C 180,E1 -13529.68,E2 -13529.68} C_VEL
LIN {X 0,Y 354.799,Z 404.911,A -85,B 0,C 180,E1 -13533.703,E2 -13533.703} C_VEL
LIN {X 0,Y 354.793,Z 404.917,A -85,B 0,C 180,E1 -13536.461,E2 -13536.461} C_VEL
LIN {X 0,Y 354.818,Z 404.908,A -85,B 0,C 180,E1 -13539.425,E2 -13539.425} C_VEL
LIN {X 0,Y 354.783,Z 404.916,A -85,B 0,C 180,E1 -13542.869,E2 -13542.869} C_VEL
LIN {X 0,Y 354.773,Z 404.916,A -85,B 0,C 180,E1 -13546.107,E2 -13546.107} C_VEL
LIN {X 0,Y 354.82,Z 404.909,A -85,B 0,C 180,E1 -13549.186,E2 -13549.186} C_VEL
LIN {X 0,Y 354.81,Z 404.915,A -85,B 0,C 180,E1 -13552.403,E2 -13552.403} C_VEL
LIN {X 0,Y 354.81,Z 404.911,A -85,B 0,C 180,E1 -13554.943,E2 -13554.943} C_VEL
LIN {X 0,Y 354.792,Z 404.918,A -85,B 0,C 180,E1 -13558.407,E2 -13558.407} C_VEL
LIN {X 0,Y 354.845,Z 404.906,A -85,B 0,C 180,E1 -13561.62,E2 -13561.62} C_VEL
LIN {X 0,Y 354.899,Z 404.903,A -85,B 0,C 180,E1 -13564.174,E2 -13564.174} C_VEL
LIN {X 0,Y 354.835,Z 404.909,A -85,B 0,C 180,E1 -13567.896,E2 -13567.896} C_VEL
LIN {X 0,Y 354.923,Z 404.897,A -85,B 0,C 180,E1 -13571.893,E2 -13571.893} C_VEL
LIN {X 0,Y 354.89,Z 404.899,A -85,B 0,C 180,E1 -13573.047,E2 -13573.047} C_VEL
LIN {X 0,Y 359.871,Z 419.186,A -85,B 0,C 180,E1 -13573.864,E2 -13573.864} C_VEL
LIN {X 0,Y 361.882,Z 425.645,A -85,B 0,C 180,E1 -13574.315,E2 -13574.315} C_VEL
LIN {X 0,Y 361.698,Z 435.963,A -85,B 0,C 180,E1 -13574.981,E2 -13574.981} C_VEL
LIN {X 0,Y 361.036,Z 447.388,A -85,B 0,C 180,E1 -13575.918,E2 -13575.918} C_VEL
LIN {X 0,Y 360.221,Z 458.136,A -85,B 0,C 180,E1 -13577.036,E2 -13577.036} C_VEL
LIN {X 0,Y 359.388,Z 466.813,A -85,B 0,C 180,E1 -13578.143,E2 -13578.143} C_VEL
LIN {X 0,Y 358.441,Z 475.887,A -85,B 0,C 180,E1 -13579.552,E2 -13579.552} C_VEL
LIN {X 0,Y 357.587,Z 484.54,A -85,B 0,C 180,E1 -13581.24,E2 -13581.24} C_VEL
LIN {X 0,Y 356.721,Z 491.542,A -85,B 0,C 180,E1 -13582.928,E2 -13582.928} C_VEL
LIN {X 0,Y 356.046,Z 497.918,A -85,B 0,C 180,E1 -13584.905,E2 -13584.905} C_VEL
LIN {X 0,Y 355.554,Z 502.119,A -85,B 0,C 180,E1 -13586.602,E2 -13586.602} C_VEL
LIN {X 0,Y 355.275,Z 504.339,A -85,B 0,C 180,E1 -13587.734,E2 -13587.734} C_VEL
LIN {X 0,Y 355.078,Z 506.144,A -85,B 0,C 180,E1 -13588.867,E2 -13588.867} C_VEL
LIN {X 0,Y 354.905,Z 508.452,A -85,B 0,C 180,E1 -13591.136,E2 -13591.136} C_VEL
LIN {X 0,Y 354.854,Z 509.045,A -85,B 0,C 180,E1 -13592.271,E2 -13592.271} C_VEL
LIN {X 0,Y 354.716,Z 509.275,A -85,B 0,C 180,E1 -13593.409,E2 -13593.409} C_VEL
LIN {X 0,Y 355.036,Z 508.455,A -85,B 0,C 180,E1 -13595.681,E2 -13595.681} C_VEL
LIN {X 0,Y 355.358,Z 507.472,A -85,B 0,C 180,E1 -13596.816,E2 -13596.816} C_VEL
LIN {X 0,Y 355.77,Z 504.478,A -85,B 0,C 180,E1 -13598.987,E2 -13598.987} C_VEL
LIN {X 0,Y 356.411,Z 500.741,A -85,B 0,C 180,E1 -13600.798,E2 -13600.798} C_VEL
LIN {X 0,Y 357.026,Z 496.11,A -85,B 0,C 180,E1 -13602.507,E2 -13602.507} C_VEL
LIN {X 0,Y 357.805,Z 490.231,A -85,B 0,C 180,E1 -13604.214,E2 -13604.214} C_VEL
LIN {X 0,Y 358.753,Z 482.87,A -85,B 0,C 180,E1 -13605.919,E2 -13605.919} C_VEL
LIN {X 0,Y 359.973,Z 473.555,A -85,B 0,C 180,E1 -13607.616,E2 -13607.616} C_VEL
LIN {X 0,Y 361.011,Z 463.936,A -85,B 0,C 180,E1 -13609.032,E2 -13609.032} C_VEL
LIN {X 0,Y 361.978,Z 453.047,A -85,B 0,C 180,E1 -13610.308,E2 -13610.308} C_VEL
LIN {X 0,Y 362.851,Z 441.073,A -85,B 0,C 180,E1 -13611.412,E2 -13611.412} C_VEL
LIN {X 0,Y 363.574,Z 429.225,A -85,B 0,C 180,E1 -13612.231,E2 -13612.231} C_VEL
LIN {X 0,Y 360.508,Z 419.536,A -85,B 0,C 180,E1 -13612.976,E2 -13612.976} C_VEL
LIN {X 0,Y 355.723,Z 407.495,A -85,B 0,C 180,E1 -13613.759,E2 -13613.759} C_VEL
LIN {X 0,Y 354.881,Z 404.903,A -85,B 0,C 180,E1 -13613.915,E2 -13613.915} C_VEL
LIN {X 0,Y 354.89,Z 404.905,A -85,B 0,C 180,E1 -13617.097,E2 -13617.097} C_VEL
LIN {X 0,Y 354.86,Z 404.909,A -85,B 0,C 180,E1 -13619.679,E2 -13619.679} C_VEL
LIN {X 0,Y 354.812,Z 404.916,A -85,B 0,C 180,E1 -13623.702,E2 -13623.702} C_VEL
LIN {X 0,Y 354.803,Z 404.915,A -85,B 0,C 180,E1 -13626.327,E2 -13626.327} C_VEL
LIN {X 0,Y 354.129,Z 404.999,A -85,B 0,C 180,E1 -13627.275,E2 -13627.275} C_VEL
LIN {X 0,Y 351.24,Z 405.356,A -85,B 0,C 180,E1 -13628.815,E2 -13628.815} C_VEL
LIN {X 0,Y 348.814,Z 405.657,A -85,B 0,C 180,E1 -13630.062,E2 -13630.062} C_VEL
LIN {X 0,Y 347.804,Z 405.786,A -85,B 0,C 180,E1 -13631.027,E2 -13631.027} C_VEL
LIN {X 0,Y 347.739,Z 405.791,A -85,B 0,C 180,E1 -13631.354,E2 -13631.354} C_VEL
LIN {X 0,Y 347.714,Z 405.793,A -85,B 0,C 180,E1 -13635.026,E2 -13635.026} C_VEL
LIN {X 0,Y 347.759,Z 405.788,A -85,B 0,C 180,E1 -13638.397,E2 -13638.397} C_VEL
LIN {X 0,Y 347.779,Z 405.762,A -85,B 0,C 180,E1 -13642.011,E2 -13642.011} C_VEL
LIN {X 0,Y 347.75,Z 405.793,A -85,B 0,C 180,E1 -13645.536,E2 -13645.536} C_VEL
LIN {X 0,Y 347.75,Z 405.773,A -85,B 0,C 180,E1 -13648.3,E2 -13648.3} C_VEL
LIN {X 0,Y 347.783,Z 405.751,A -85,B 0,C 180,E1 -13650.988,E2 -13650.988} C_VEL
LIN {X 0,Y 347.835,Z 405.773,A -85,B 0,C 180,E1 -13653.608,E2 -13653.608} C_VEL
LIN {X 0,Y 347.79,Z 405.789,A -85,B 0,C 180,E1 -13656.162,E2 -13656.162} C_VEL
LIN {X 0,Y 347.836,Z 405.964,A -85,B 0,C 180,E1 -13658.754,E2 -13658.754} C_VEL
LIN {X 0,Y 351.728,Z 419.121,A -85,B 0,C 180,E1 -13659.907,E2 -13659.907} C_VEL
LIN {X 0,Y 354.635,Z 429.249,A -85,B 0,C 180,E1 -13660.935,E2 -13660.935} C_VEL
LIN {X 0,Y 353.706,Z 441.882,A -85,B 0,C 180,E1 -13662.212,E2 -13662.212} C_VEL
LIN {X 0,Y 352.544,Z 454.749,A -85,B 0,C 180,E1 -13663.794,E2 -13663.794} C_VEL
LIN {X 0,Y 351.344,Z 466.302,A -85,B 0,C 180,E1 -13665.52,E2 -13665.52} C_VEL
LIN {X 0,Y 350.456,Z 475.852,A -85,B 0,C 180,E1 -13667.256,E2 -13667.256} C_VEL
LIN {X 0,Y 349.568,Z 485.06,A -85,B 0,C 180,E1 -13669.282,E2 -13669.282} C_VEL
LIN {X 0,Y 348.926,Z 492.578,A -85,B 0,C 180,E1 -13671.311,E2 -13671.311} C_VEL
LIN {X 0,Y 348.396,Z 499.415,A -85,B 0,C 180,E1 -13673.63,E2 -13673.63} C_VEL
LIN {X 0,Y 347.902,Z 503.421,A -85,B 0,C 180,E1 -13675.365,E2 -13675.365} C_VEL
LIN {X 0,Y 347.857,Z 507.455,A -85,B 0,C 180,E1 -13677.684,E2 -13677.684} C_VEL
LIN {X 0,Y 347.917,Z 510.088,A -85,B 0,C 180,E1 -13680,E2 -13680} C_VEL
LIN {X 0,Y 348.142,Z 511.336,A -85,B 0,C 180,E1 -13682.314,E2 -13682.314} C_VEL
LIN {X 0,Y 348.507,Z 511.242,A -85,B 0,C 180,E1 -13684.626,E2 -13684.626} C_VEL
LIN {X 0,Y 349.097,Z 509.829,A -85,B 0,C 180,E1 -13686.938,E2 -13686.938} C_VEL
LIN {X 0,Y 350.027,Z 507.043,A -85,B 0,C 180,E1 -13689.243,E2 -13689.243} C_VEL
LIN {X 0,Y 351.257,Z 502.828,A -85,B 0,C 180,E1 -13691.541,E2 -13691.541} C_VEL
LIN {X 0,Y 352.313,Z 498.639,A -85,B 0,C 180,E1 -13693.262,E2 -13693.262} C_VEL
LIN {X 0,Y 354.087,Z 491.585,A -85,B 0,C 180,E1 -13695.542,E2 -13695.542} C_VEL
LIN {X 0,Y 355.959,Z 483.732,A -85,B 0,C 180,E1 -13697.523,E2 -13697.523} C_VEL
LIN {X 0,Y 358.124,Z 474.078,A -85,B 0,C 180,E1 -13699.488,E2 -13699.488} C_VEL
LIN {X 0,Y 360.127,Z 464.082,A -85,B 0,C 180,E1 -13701.163,E2 -13701.163} C_VEL
LIN {X 0,Y 362.197,Z 453.007,A -85,B 0,C 180,E1 -13702.684,E2 -13702.684} C_VEL
LIN {X 0,Y 363.994,Z 442.136,A -85,B 0,C 180,E1 -13703.92,E2 -13703.92} C_VEL
LIN {X 0,Y 363.489,Z 439.228,A -85,B 0,C 180,E1 -13704.355,E2 -13704.355} C_VEL
LIN {X 0,Y 360.469,Z 429.96,A -85,B 0,C 180,E1 -13705.876,E2 -13705.876} C_VEL
LIN {X 0,Y 356.428,Z 421.094,A -85,B 0,C 180,E1 -13707.462,E2 -13707.462} C_VEL
LIN {X 0,Y 352.07,Z 413.468,A -85,B 0,C 180,E1 -13708.995,E2 -13708.995} C_VEL
LIN {X 0,Y 350.644,Z 410.65,A -85,B 0,C 180,E1 -13709.536,E2 -13709.536} C_VEL
LIN {X 0,Y 348.444,Z 408.092,A -85,B 0,C 180,E1 -13710.225,E2 -13710.225} C_VEL
LIN {X 0,Y 347.77,Z 405.789,A -85,B 0,C 180,E1 -13710.598,E2 -13710.598} C_VEL
LIN {X 0,Y 348.173,Z 407.687,A -85,B 0,C 180,E1 -13714.146,E2 -13714.146} C_VEL
LIN {X 0,Y 348.698,Z 410.106,A -85,B 0,C 180,E1 -13717.203,E2 -13717.203} C_VEL
LIN {X 0,Y 349.369,Z 413.14,A -85,B 0,C 180,E1 -13720.144,E2 -13720.144} C_VEL
LIN {X 0,Y 350.411,Z 417.924,A -85,B 0,C 180,E1 -13723.776,E2 -13723.776} C_VEL
LIN {X 0,Y 351.525,Z 423.522,A -85,B 0,C 180,E1 -13727.174,E2 -13727.174} C_VEL
LIN {X 0,Y 352.174,Z 427.649,A -85,B 0,C 180,E1 -13729.317,E2 -13729.317} C_VEL
LIN {X 0,Y 351.732,Z 431.082,A -85,B 0,C 180,E1 -13730.836,E2 -13730.836} C_VEL
LIN {X 0,Y 350.031,Z 441.519,A -85,B 0,C 180,E1 -13734.993,E2 -13734.993} C_VEL
LIN {X 0,Y 349.067,Z 450.938,A -85,B 0,C 180,E1 -13738.433,E2 -13738.433} C_VEL
LIN {X 0,Y 348.629,Z 456.635,A -85,B 0,C 180,E1 -13740.377,E2 -13740.377} C_VEL
LIN {X 0,Y 349.641,Z 461.187,A -85,B 0,C 180,E1 -13740.826,E2 -13740.826} C_VEL
LIN {X 0,Y 350.449,Z 463.947,A -85,B 0,C 180,E1 -13741.131,E2 -13741.131} C_VEL
LIN {X 0,Y 353.076,Z 475.032,A -85,B 0,C 180,E1 -13742.24,E2 -13742.24} C_VEL
LIN {X 0,Y 355.413,Z 488.874,A -85,B 0,C 180,E1 -13743.551,E2 -13743.551} C_VEL
LIN {X 0,Y 356.564,Z 503.91,A -85,B 0,C 180,E1 -13744.93,E2 -13744.93} C_VEL
LIN {X 0,Y 356.269,Z 517.143,A -85,B 0,C 180,E1 -13746.166,E2 -13746.166} C_VEL
LIN {X 0,Y 355.319,Z 531.112,A -85,B 0,C 180,E1 -13747.619,E2 -13747.619} C_VEL
LIN {X 0,Y 354.687,Z 537.789,A -85,B 0,C 180,E1 -13748.388,E2 -13748.388} C_VEL
LIN {X 0,Y 352.2,Z 551.799,A -85,B 0,C 180,E1 -13750.169,E2 -13750.169} C_VEL
LIN {X 0,Y 350.461,Z 562.997,A -85,B 0,C 180,E1 -13751.89,E2 -13751.89} C_VEL
LIN {X 0,Y 349.045,Z 572.577,A -85,B 0,C 180,E1 -13753.626,E2 -13753.626} C_VEL
LIN {X 0,Y 347.887,Z 582.198,A -85,B 0,C 180,E1 -13755.701,E2 -13755.701} C_VEL
LIN {X 0,Y 347.213,Z 589.98,A -85,B 0,C 180,E1 -13757.728,E2 -13757.728} C_VEL
LIN {X 0,Y 346.921,Z 595.615,A -85,B 0,C 180,E1 -13759.494,E2 -13759.494} C_VEL
LIN {X 0,Y 346.854,Z 601.674,A -85,B 0,C 180,E1 -13761.845,E2 -13761.845} C_VEL
LIN {X 0,Y 346.991,Z 604.691,A -85,B 0,C 180,E1 -13763.318,E2 -13763.318} C_VEL
LIN {X 0,Y 347.252,Z 607.811,A -85,B 0,C 180,E1 -13765.355,E2 -13765.355} C_VEL
LIN {X 0,Y 347.313,Z 609.079,A -85,B 0,C 180,E1 -13766.518,E2 -13766.518} C_VEL
LIN {X 0,Y 347.602,Z 610.496,A -85,B 0,C 180,E1 -13768.84,E2 -13768.84} C_VEL
LIN {X 0,Y 347.79,Z 610.638,A -85,B 0,C 180,E1 -13769.999,E2 -13769.999} C_VEL
LIN {X 0,Y 347.451,Z 609.656,A -85,B 0,C 180,E1 -13772.317,E2 -13772.317} C_VEL
LIN {X 0,Y 347.314,Z 607.159,A -85,B 0,C 180,E1 -13774.641,E2 -13774.641} C_VEL
LIN {X 0,Y 347.156,Z 604.256,A -85,B 0,C 180,E1 -13776.392,E2 -13776.392} C_VEL
LIN {X 0,Y 347.045,Z 600.334,A -85,B 0,C 180,E1 -13778.148,E2 -13778.148} C_VEL
LIN {X 0,Y 347.066,Z 595.403,A -85,B 0,C 180,E1 -13779.91,E2 -13779.91} C_VEL
LIN {X 0,Y 347.322,Z 588.249,A -85,B 0,C 180,E1 -13781.969,E2 -13781.969} C_VEL
LIN {X 0,Y 347.876,Z 579.372,A -85,B 0,C 180,E1 -13784.029,E2 -13784.029} C_VEL
LIN {X 0,Y 348.701,Z 570.091,A -85,B 0,C 180,E1 -13785.787,E2 -13785.787} C_VEL
LIN {X 0,Y 349.891,Z 558.86,A -85,B 0,C 180,E1 -13787.534,E2 -13787.534} C_VEL
LIN {X 0,Y 351.238,Z 546.332,A -85,B 0,C 180,E1 -13789.125,E2 -13789.125} C_VEL
LIN {X 0,Y 352.561,Z 533.83,A -85,B 0,C 180,E1 -13790.416,E2 -13790.416} C_VEL
LIN {X 0,Y 352.717,Z 528.551,A -85,B 0,C 180,E1 -13790.893,E2 -13790.893} C_VEL
LIN {X 0,Y 351.691,Z 514.859,A -85,B 0,C 180,E1 -13792.004,E2 -13792.004} C_VEL
LIN {X 0,Y 350.335,Z 501.413,A -85,B 0,C 180,E1 -13792.89,E2 -13792.89} C_VEL
LIN {X 0,Y 348.648,Z 485.731,A -85,B 0,C 180,E1 -13793.68,E2 -13793.68} C_VEL
LIN {X 0,Y 347.902,Z 478.655,A -85,B 0,C 180,E1 -13793.99,E2 -13793.99} C_VEL
LIN {X 0,Y 348.823,Z 465.986,A -85,B 0,C 180,E1 -13798.258,E2 -13798.258} C_VEL
LIN {X 0,Y 349.902,Z 455.052,A -85,B 0,C 180,E1 -13802.002,E2 -13802.002} C_VEL
LIN {X 0,Y 351.006,Z 444.984,A -85,B 0,C 180,E1 -13805.494,E2 -13805.494} C_VEL
LIN {X 0,Y 352.463,Z 433.293,A -85,B 0,C 180,E1 -13809.646,E2 -13809.646} C_VEL
LIN {X 0,Y 352.47,Z 429.24,A -85,B 0,C 180,E1 -13811.145,E2 -13811.145} C_VEL
LIN {X 0,Y 351.086,Z 422.278,A -85,B 0,C 180,E1 -13813.893,E2 -13813.893} C_VEL
LIN {X 0,Y 349.284,Z 413.266,A -85,B 0,C 180,E1 -13817.603,E2 -13817.603} C_VEL
LIN {X 0,Y 347.784,Z 405.791,A -85,B 0,C 180,E1 -13820.924,E2 -13820.924} C_VEL
LIN {X 0,Y 347.78,Z 405.786,A -85,B 0,C 180,E1 -13824.124,E2 -13824.124} C_VEL
LIN {X 0,Y 347.729,Z 405.792,A -85,B 0,C 180,E1 -13828.085,E2 -13828.085} C_VEL
LIN {X 0,Y 347.797,Z 405.788,A -85,B 0,C 180,E1 -13830.99,E2 -13830.99} C_VEL
LIN {X 0,Y 347.822,Z 405.782,A -85,B 0,C 180,E1 -13833.607,E2 -13833.607} C_VEL
LIN {X 0,Y 347.778,Z 405.786,A -85,B 0,C 180,E1 -13836.161,E2 -13836.161} C_VEL
LIN {X 0,Y 347.802,Z 405.782,A -85,B 0,C 180,E1 -13839.909,E2 -13839.909} C_VEL
LIN {X 0,Y 347.856,Z 405.777,A -85,B 0,C 180,E1 -13842.359,E2 -13842.359} C_VEL
LIN {X 0,Y 347.887,Z 405.772,A -85,B 0,C 180,E1 -13845.971,E2 -13845.971} C_VEL
LIN {X 0,Y 347.923,Z 405.768,A -85,B 0,C 180,E1 -13849.526,E2 -13849.526} C_VEL
LIN {X 0,Y 348.063,Z 405.75,A -85,B 0,C 180,E1 -13851.875,E2 -13851.875} C_VEL
LIN {X 0,Y 348.058,Z 405.751,A -85,B 0,C 180,E1 -13854.206,E2 -13854.206} C_VEL
LIN {X 0,Y 348.198,Z 405.734,A -85,B 0,C 180,E1 -13857.687,E2 -13857.687} C_VEL
LIN {X 0,Y 348.358,Z 405.713,A -85,B 0,C 180,E1 -13860,E2 -13860} C_VEL
LIN {X 0,Y 348.199,Z 405.734,A -85,B 0,C 180,E1 -13862.314,E2 -13862.314} C_VEL
LIN {X 0,Y 348.096,Z 405.749,A -85,B 0,C 180,E1 -13866.958,E2 -13866.958} C_VEL
LIN {X 0,Y 347.959,Z 405.763,A -85,B 0,C 180,E1 -13869.299,E2 -13869.299} C_VEL
LIN {X 0,Y 347.884,Z 405.778,A -85,B 0,C 180,E1 -13872.84,E2 -13872.84} C_VEL
LIN {X 0,Y 347.83,Z 405.782,A -85,B 0,C 180,E1 -13876.432,E2 -13876.432} C_VEL
LIN {X 0,Y 347.846,Z 405.782,A -85,B 0,C 180,E1 -13878.861,E2 -13878.861} C_VEL
LIN {X 0,Y 347.765,Z 405.792,A -85,B 0,C 180,E1 -13882.58,E2 -13882.58} C_VEL
LIN {X 0,Y 347.804,Z 405.785,A -85,B 0,C 180,E1 -13885.11,E2 -13885.11} C_VEL
LIN {X 0,Y 347.803,Z 405.782,A -85,B 0,C 180,E1 -13887.695,E2 -13887.695} C_VEL
LIN {X 0,Y 347.756,Z 405.789,A -85,B 0,C 180,E1 -13890.348,E2 -13890.348} C_VEL
LIN {X 0,Y 347.737,Z 405.795,A -85,B 0,C 180,E1 -13894.465,E2 -13894.465} C_VEL
LIN {X 0,Y 347.768,Z 405.786,A -85,B 0,C 180,E1 -13897.99,E2 -13897.99} C_VEL
LIN {X 0,Y 347.745,Z 405.79,A -85,B 0,C 180,E1 -13901.832,E2 -13901.832} C_VEL
LIN {X 0,Y 347.761,Z 405.788,A -85,B 0,C 180,E1 -13905.018,E2 -13905.018} C_VEL
LIN {X 0,Y 347.764,Z 405.793,A -85,B 0,C 180,E1 -13908.395,E2 -13908.395} C_VEL
LIN {X 0,Y 347.776,Z 405.787,A -85,B 0,C 180,E1 -13912.012,E2 -13912.012} C_VEL
LIN {X 0,Y 347.742,Z 405.79,A -85,B 0,C 180,E1 -13915.538,E2 -13915.538} C_VEL
LIN {X 0,Y 347.759,Z 405.788,A -85,B 0,C 180,E1 -13919.655,E2 -13919.655} C_VEL
LIN {X 0,Y 347.83,Z 405.78,A -85,B 0,C 180,E1 -13923.609,E2 -13923.609} C_VEL
LIN {X 0,Y 347.789,Z 405.789,A -85,B 0,C 180,E1 -13926.164,E2 -13926.164} C_VEL
LIN {X 0,Y 347.813,Z 405.785,A -85,B 0,C 180,E1 -13929.911,E2 -13929.911} C_VEL
LIN {X 0,Y 347.847,Z 405.773,A -85,B 0,C 180,E1 -13932.656,E2 -13932.656} C_VEL
LIN {X 0,Y 352.628,Z 419.334,A -85,B 0,C 180,E1 -13933.442,E2 -13933.442} C_VEL
LIN {X 0,Y 355.149,Z 427.167,A -85,B 0,C 180,E1 -13934.006,E2 -13934.006} C_VEL
LIN {X 0,Y 355.026,Z 436.016,A -85,B 0,C 180,E1 -13934.585,E2 -13934.585} C_VEL
LIN {X 0,Y 354.359,Z 447.252,A -85,B 0,C 180,E1 -13935.501,E2 -13935.501} C_VEL
LIN {X 0,Y 353.503,Z 458.212,A -85,B 0,C 180,E1 -13936.639,E2 -13936.639} C_VEL
LIN {X 0,Y 352.557,Z 468.062,A -85,B 0,C 180,E1 -13937.91,E2 -13937.91} C_VEL
LIN {X 0,Y 351.555,Z 477.082,A -85,B 0,C 180,E1 -13939.345,E2 -13939.345} C_VEL
LIN {X 0,Y 350.664,Z 485.703,A -85,B 0,C 180,E1 -13941.066,E2 -13941.066} C_VEL
LIN {X 0,Y 349.766,Z 492.678,A -85,B 0,C 180,E1 -13942.787,E2 -13942.787} C_VEL
LIN {X 0,Y 349.251,Z 497.372,A -85,B 0,C 180,E1 -13944.227,E2 -13944.227} C_VEL
LIN {X 0,Y 348.748,Z 501.921,A -85,B 0,C 180,E1 -13945.957,E2 -13945.957} C_VEL
LIN {X 0,Y 348.258,Z 505.407,A -85,B 0,C 180,E1 -13947.688,E2 -13947.688} C_VEL
LIN {X 0,Y 348.056,Z 507.198,A -85,B 0,C 180,E1 -13948.844,E2 -13948.844} C_VEL
LIN {X 0,Y 347.893,Z 509.479,A -85,B 0,C 180,E1 -13951.159,E2 -13951.159} C_VEL
LIN {X 0,Y 347.829,Z 510.064,A -85,B 0,C 180,E1 -13952.317,E2 -13952.317} C_VEL
LIN {X 0,Y 347.692,Z 510.277,A -85,B 0,C 180,E1 -13953.478,E2 -13953.478} C_VEL
LIN {X 0,Y 348.037,Z 509.435,A -85,B 0,C 180,E1 -13955.796,E2 -13955.796} C_VEL
LIN {X 0,Y 348.374,Z 508.442,A -85,B 0,C 180,E1 -13956.953,E2 -13956.953} C_VEL
LIN {X 0,Y 348.829,Z 505.417,A -85,B 0,C 180,E1 -13959.166,E2 -13959.166} C_VEL
LIN {X 0,Y 349.503,Z 501.656,A -85,B 0,C 180,E1 -13961.014,E2 -13961.014} C_VEL
LIN {X 0,Y 350.14,Z 497.003,A -85,B 0,C 180,E1 -13962.757,E2 -13962.757} C_VEL
LIN {X 0,Y 350.964,Z 491.098,A -85,B 0,C 180,E1 -13964.497,E2 -13964.497} C_VEL
LIN {X 0,Y 351.974,Z 483.691,A -85,B 0,C 180,E1 -13966.234,E2 -13966.234} C_VEL
LIN {X 0,Y 353.253,Z 474.337,A -85,B 0,C 180,E1 -13967.962,E2 -13967.962} C_VEL
LIN {X 0,Y 354.355,Z 464.658,A -85,B 0,C 180,E1 -13969.404,E2 -13969.404} C_VEL
LIN {X 0,Y 355.368,Z 453.692,A -85,B 0,C 180,E1 -13970.703,E2 -13970.703} C_VEL
LIN {X 0,Y 356.251,Z 441.972,A -85,B 0,C 180,E1 -13971.798,E2 -13971.798} C_VEL
LIN {X 0,Y 356.805,Z 430.028,A -85,B 0,C 180,E1 -13972.649,E2 -13972.649} C_VEL
LIN {X 0,Y 352.741,Z 418.213,A -85,B 0,C 180,E1 -13973.579,E2 -13973.579} C_VEL
LIN {X 0,Y 347.874,Z 406.097,A -85,B 0,C 180,E1 -13974.354,E2 -13974.354} C_VEL
LIN {X 0,Y 347.834,Z 405.779,A -85,B 0,C 180,E1 -13974.471,E2 -13974.471} C_VEL
LIN {X 0,Y 347.817,Z 405.785,A -85,B 0,C 180,E1 -13977.694,E2 -13977.694} C_VEL
LIN {X 0,Y 347.77,Z 405.794,A -85,B 0,C 180,E1 -13980.347,E2 -13980.347} C_VEL
LIN {X 0,Y 347.75,Z 405.795,A -85,B 0,C 180,E1 -13984.464,E2 -13984.464} C_VEL
LIN {X 0,Y 347.779,Z 405.776,A -85,B 0,C 180,E1 -13987.989,E2 -13987.989} C_VEL
LIN {X 0,Y 347.739,Z 405.791,A -85,B 0,C 180,E1 -13991.354,E2 -13991.354} C_VEL
LIN {X 0,Y 347.108,Z 405.873,A -85,B 0,C 180,E1 -13992.321,E2 -13992.321} C_VEL
LIN {X 0,Y 344.239,Z 406.231,A -85,B 0,C 180,E1 -13993.893,E2 -13993.893} C_VEL
LIN {X 0,Y 341.787,Z 406.533,A -85,B 0,C 180,E1 -13995.165,E2 -13995.165} C_VEL
LIN {X 0,Y 340.741,Z 406.662,A -85,B 0,C 180,E1 -13996.151,E2 -13996.151} C_VEL
LIN {X 0,Y 340.661,Z 406.672,A -85,B 0,C 180,E1 -13996.485,E2 -13996.485} C_VEL
LIN {X 0,Y 340.696,Z 406.653,A -85,B 0,C 180,E1 -13999.753,E2 -13999.753} C_VEL
LIN {X 0,Y 340.711,Z 406.659,A -85,B 0,C 180,E1 -14003.259,E2 -14003.259} C_VEL
LIN {X 0,Y 340.699,Z 406.67,A -85,B 0,C 180,E1 -14006.154,E2 -14006.154} C_VEL
LIN {X 0,Y 340.746,Z 406.624,A -85,B 0,C 180,E1 -14010.329,E2 -14010.329} C_VEL
LIN {X 0,Y 340.808,Z 406.644,A -85,B 0,C 180,E1 -14013.02,E2 -14013.02} C_VEL
LIN {X 0,Y 340.759,Z 406.666,A -85,B 0,C 180,E1 -14015.638,E2 -14015.638} C_VEL
LIN {X 0,Y 340.739,Z 406.666,A -85,B 0,C 180,E1 -14018.422,E2 -14018.422} C_VEL
LIN {X 0,Y 345.276,Z 422.072,A -85,B 0,C 180,E1 -14019.82,E2 -14019.82} C_VEL
LIN {X 0,Y 347.805,Z 430.926,A -85,B 0,C 180,E1 -14020.754,E2 -14020.754} C_VEL
LIN {X 0,Y 346.654,Z 444.247,A -85,B 0,C 180,E1 -14022.143,E2 -14022.143} C_VEL
LIN {X 0,Y 345.589,Z 455.799,A -85,B 0,C 180,E1 -14023.61,E2 -14023.61} C_VEL
LIN {X 0,Y 344.441,Z 466.427,A -85,B 0,C 180,E1 -14025.223,E2 -14025.223} C_VEL
LIN {X 0,Y 343.533,Z 476.149,A -85,B 0,C 180,E1 -14026.995,E2 -14026.995} C_VEL
LIN {X 0,Y 342.591,Z 485.487,A -85,B 0,C 180,E1 -14029.061,E2 -14029.061} C_VEL
LIN {X 0,Y 341.873,Z 493.631,A -85,B 0,C 180,E1 -14031.288,E2 -14031.288} C_VEL
LIN {X 0,Y 341.39,Z 500.088,A -85,B 0,C 180,E1 -14033.498,E2 -14033.498} C_VEL
LIN {X 0,Y 340.877,Z 504.209,A -85,B 0,C 180,E1 -14035.269,E2 -14035.269} C_VEL
LIN {X 0,Y 340.715,Z 506.48,A -85,B 0,C 180,E1 -14036.452,E2 -14036.452} C_VEL
LIN {X 0,Y 340.887,Z 509.897,A -85,B 0,C 180,E1 -14038.818,E2 -14038.818} C_VEL
LIN {X 0,Y 340.973,Z 511.968,A -85,B 0,C 180,E1 -14041.181,E2 -14041.181} C_VEL
LIN {X 0,Y 341.323,Z 512.664,A -85,B 0,C 180,E1 -14043.541,E2 -14043.541} C_VEL
LIN {X 0,Y 341.827,Z 512.025,A -85,B 0,C 180,E1 -14045.9,E2 -14045.9} C_VEL
LIN {X 0,Y 342.653,Z 510.046,A -85,B 0,C 180,E1 -14048.254,E2 -14048.254} C_VEL
LIN {X 0,Y 343.838,Z 506.675,A -85,B 0,C 180,E1 -14050.6,E2 -14050.6} C_VEL
LIN {X 0,Y 345.203,Z 501.874,A -85,B 0,C 180,E1 -14052.941,E2 -14052.941} C_VEL
LIN {X 0,Y 346.531,Z 497.178,A -85,B 0,C 180,E1 -14054.685,E2 -14054.685} C_VEL
LIN {X 0,Y 348.341,Z 490.444,A -85,B 0,C 180,E1 -14056.708,E2 -14056.708} C_VEL
LIN {X 0,Y 350.477,Z 482.13,A -85,B 0,C 180,E1 -14058.714,E2 -14058.714} C_VEL
LIN {X 0,Y 352.797,Z 472.031,A -85,B 0,C 180,E1 -14060.676,E2 -14060.676} C_VEL
LIN {X 0,Y 355.106,Z 461.201,A -85,B 0,C 180,E1 -14062.394,E2 -14062.394} C_VEL
LIN {X 0,Y 357.266,Z 450.067,A -85,B 0,C 180,E1 -14063.848,E2 -14063.848} C_VEL
LIN {X 0,Y 358.242,Z 444.516,A -85,B 0,C 180,E1 -14064.476,E2 -14064.476} C_VEL
LIN {X 0,Y 355.693,Z 435.254,A -85,B 0,C 180,E1 -14066.067,E2 -14066.067} C_VEL
LIN {X 0,Y 352.137,Z 426.67,A -85,B 0,C 180,E1 -14067.683,E2 -14067.683} C_VEL
LIN {X 0,Y 348.297,Z 419.331,A -85,B 0,C 180,E1 -14069.219,E2 -14069.219} C_VEL
LIN {X 0,Y 346.238,Z 415.767,A -85,B 0,C 180,E1 -14070.028,E2 -14070.028} C_VEL
LIN {X 0,Y 344.549,Z 413.379,A -85,B 0,C 180,E1 -14070.66,E2 -14070.66} C_VEL
LIN {X 0,Y 343.813,Z 411.763,A -85,B 0,C 180,E1 -14070.99,E2 -14070.99} C_VEL
LIN {X 0,Y 341.77,Z 409.958,A -85,B 0,C 180,E1 -14071.682,E2 -14071.682} C_VEL
LIN {X 0,Y 341.113,Z 408.626,A -85,B 0,C 180,E1 -14072.041,E2 -14072.041} C_VEL
LIN {X 0,Y 341.578,Z 410.637,A -85,B 0,C 180,E1 -14075.177,E2 -14075.177} C_VEL
LIN {X 0,Y 342.276,Z 413.756,A -85,B 0,C 180,E1 -14078.714,E2 -14078.714} C_VEL
LIN {X 0,Y 342.811,Z 416.33,A -85,B 0,C 180,E1 -14080.998,E2 -14080.998} C_VEL
LIN {X 0,Y 343.81,Z 420.845,A -85,B 0,C 180,E1 -14084.319,E2 -14084.319} C_VEL
LIN {X 0,Y 344.891,Z 426.544,A -85,B 0,C 180,E1 -14087.742,E2 -14087.742} C_VEL
LIN {X 0,Y 345.305,Z 429.659,A -85,B 0,C 180,E1 -14089.359,E2 -14089.359} C_VEL
LIN {X 0,Y 344.799,Z 432.883,A -85,B 0,C 180,E1 -14090.811,E2 -14090.811} C_VEL
LIN {X 0,Y 343.055,Z 443.255,A -85,B 0,C 180,E1 -14095.031,E2 -14095.031} C_VEL
LIN {X 0,Y 341.913,Z 453.768,A -85,B 0,C 180,E1 -14098.948,E2 -14098.948} C_VEL
LIN {X 0,Y 342.914,Z 458.359,A -85,B 0,C 180,E1 -14099.468,E2 -14099.468} C_VEL
LIN {X 0,Y 343.843,Z 461.219,A -85,B 0,C 180,E1 -14099.84,E2 -14099.84} C_VEL
LIN {X 0,Y 347.451,Z 476.836,A -85,B 0,C 180,E1 -14101.566,E2 -14101.566} C_VEL
LIN {X 0,Y 349.579,Z 491.326,A -85,B 0,C 180,E1 -14103.033,E2 -14103.033} C_VEL
LIN {X 0,Y 350.4,Z 506.234,A -85,B 0,C 180,E1 -14104.498,E2 -14104.498} C_VEL
LIN {X 0,Y 349.797,Z 519.621,A -85,B 0,C 180,E1 -14105.834,E2 -14105.834} C_VEL
LIN {X 0,Y 348.672,Z 532.968,A -85,B 0,C 180,E1 -14107.325,E2 -14107.325} C_VEL
LIN {X 0,Y 347.754,Z 540.148,A -85,B 0,C 180,E1 -14108.2,E2 -14108.2} C_VEL
LIN {X 0,Y 345.509,Z 551.841,A -85,B 0,C 180,E1 -14109.768,E2 -14109.768} C_VEL
LIN {X 0,Y 343.387,Z 564.433,A -85,B 0,C 180,E1 -14111.812,E2 -14111.812} C_VEL
LIN {X 0,Y 341.757,Z 574.969,A -85,B 0,C 180,E1 -14113.881,E2 -14113.881} C_VEL
LIN {X 0,Y 340.569,Z 584.182,A -85,B 0,C 180,E1 -14116.063,E2 -14116.063} C_VEL
LIN {X 0,Y 340.059,Z 591.186,A -85,B 0,C 180,E1 -14118.072,E2 -14118.072} C_VEL
LIN {X 0,Y 339.769,Z 597.981,A -85,B 0,C 180,E1 -14120.474,E2 -14120.474} C_VEL
LIN {X 0,Y 339.878,Z 603.168,A -85,B 0,C 180,E1 -14122.872,E2 -14122.872} C_VEL
LIN {X 0,Y 340.18,Z 606.798,A -85,B 0,C 180,E1 -14125.259,E2 -14125.259} C_VEL
LIN {X 0,Y 340.267,Z 608.027,A -85,B 0,C 180,E1 -14126.446,E2 -14126.446} C_VEL
LIN {X 0,Y 340.577,Z 609.37,A -85,B 0,C 180,E1 -14128.816,E2 -14128.816} C_VEL
LIN {X 0,Y 340.779,Z 609.481,A -85,B 0,C 180,E1 -14129.999,E2 -14129.999} C_VEL
LIN {X 0,Y 340.615,Z 609.149,A -85,B 0,C 180,E1 -14131.181,E2 -14131.181} C_VEL
LIN {X 0,Y 340.347,Z 607.344,A -85,B 0,C 180,E1 -14133.55,E2 -14133.55} C_VEL
LIN {X 0,Y 340.285,Z 605.866,A -85,B 0,C 180,E1 -14134.737,E2 -14134.737} C_VEL
LIN {X 0,Y 340.142,Z 602.888,A -85,B 0,C 180,E1 -14136.524,E2 -14136.524} C_VEL
LIN {X 0,Y 340.01,Z 598.923,A -85,B 0,C 180,E1 -14138.318,E2 -14138.318} C_VEL
LIN {X 0,Y 340.019,Z 593.894,A -85,B 0,C 180,E1 -14140.117,E2 -14140.117} C_VEL
LIN {X 0,Y 340.276,Z 586.635,A -85,B 0,C 180,E1 -14142.221,E2 -14142.221} C_VEL
LIN {X 0,Y 340.91,Z 577.613,A -85,B 0,C 180,E1 -14144.321,E2 -14144.321} C_VEL
LIN {X 0,Y 341.777,Z 568.167,A -85,B 0,C 180,E1 -14146.116,E2 -14146.116} C_VEL
LIN {X 0,Y 342.951,Z 557.827,A -85,B 0,C 180,E1 -14147.746,E2 -14147.746} C_VEL
LIN {X 0,Y 344.324,Z 545.307,A -85,B 0,C 180,E1 -14149.369,E2 -14149.369} C_VEL
LIN {X 0,Y 345.753,Z 531.969,A -85,B 0,C 180,E1 -14150.768,E2 -14150.768} C_VEL
LIN {X 0,Y 345.033,Z 519.197,A -85,B 0,C 180,E1 -14151.9,E2 -14151.9} C_VEL
LIN {X 0,Y 343.756,Z 505.062,A -85,B 0,C 180,E1 -14152.928,E2 -14152.928} C_VEL
LIN {X 0,Y 342.124,Z 489.797,A -85,B 0,C 180,E1 -14153.798,E2 -14153.798} C_VEL
LIN {X 0,Y 340.889,Z 477.792,A -85,B 0,C 180,E1 -14154.35,E2 -14154.35} C_VEL
LIN {X 0,Y 341.718,Z 466.559,A -85,B 0,C 180,E1 -14158.23,E2 -14158.23} C_VEL
LIN {X 0,Y 342.88,Z 455.197,A -85,B 0,C 180,E1 -14162.201,E2 -14162.201} C_VEL
LIN {X 0,Y 344.002,Z 445.437,A -85,B 0,C 180,E1 -14165.676,E2 -14165.676} C_VEL
LIN {X 0,Y 345.49,Z 433.774,A -85,B 0,C 180,E1 -14169.904,E2 -14169.904} C_VEL
LIN {X 0,Y 345.497,Z 430.419,A -85,B 0,C 180,E1 -14171.18,E2 -14171.18} C_VEL
LIN {X 0,Y 343.897,Z 422.586,A -85,B 0,C 180,E1 -14174.335,E2 -14174.335} C_VEL
LIN {X 0,Y 342.071,Z 413.301,A -85,B 0,C 180,E1 -14178.251,E2 -14178.251} C_VEL
LIN {X 0,Y 340.72,Z 406.671,A -85,B 0,C 180,E1 -14181.256,E2 -14181.256} C_VEL
LIN {X 0,Y 340.71,Z 406.669,A -85,B 0,C 180,E1 -14184.72,E2 -14184.72} C_VEL
LIN {X 0,Y 340.695,Z 406.672,A -85,B 0,C 180,E1 -14188.955,E2 -14188.955} C_VEL
LIN {X 0,Y 340.77,Z 406.66,A -85,B 0,C 180,E1 -14192.473,E2 -14192.473} C_VEL
LIN {X 0,Y 340.746,Z 406.663,A -85,B 0,C 180,E1 -14195.638,E2 -14195.638} C_VEL
LIN {X 0,Y 340.735,Z 406.665,A -85,B 0,C 180,E1 -14199.474,E2 -14199.474} C_VEL
LIN {X 0,Y 340.847,Z 406.649,A -85,B 0,C 180,E1 -14201.984,E2 -14201.984} C_VEL
LIN {X 0,Y 340.859,Z 406.648,A -85,B 0,C 180,E1 -14205.705,E2 -14205.705} C_VEL
LIN {X 0,Y 340.865,Z 406.649,A -85,B 0,C 180,E1 -14209.306,E2 -14209.306} C_VEL
LIN {X 0,Y 341.065,Z 406.628,A -85,B 0,C 180,E1 -14212.898,E2 -14212.898} C_VEL
LIN {X 0,Y 341.16,Z 406.611,A -85,B 0,C 180,E1 -14217.639,E2 -14217.639} C_VEL
LIN {X 0,Y 341.307,Z 406.592,A -85,B 0,C 180,E1 -14220,E2 -14220} C_VEL
LIN {X 0,Y 341.161,Z 406.611,A -85,B 0,C 180,E1 -14222.362,E2 -14222.362} C_VEL
LIN {X 0,Y 341.066,Z 406.622,A -85,B 0,C 180,E1 -14227.102,E2 -14227.102} C_VEL
LIN {X 0,Y 340.866,Z 406.648,A -85,B 0,C 180,E1 -14230.694,E2 -14230.694} C_VEL
LIN {X 0,Y 340.853,Z 406.65,A -85,B 0,C 180,E1 -14234.326,E2 -14234.326} C_VEL
LIN {X 0,Y 340.829,Z 406.654,A -85,B 0,C 180,E1 -14238.468,E2 -14238.468} C_VEL
LIN {X 0,Y 340.745,Z 406.661,A -85,B 0,C 180,E1 -14241.858,E2 -14241.858} C_VEL
LIN {X 0,Y 340.764,Z 406.66,A -85,B 0,C 180,E1 -14245.665,E2 -14245.665} C_VEL
LIN {X 0,Y 340.733,Z 406.665,A -85,B 0,C 180,E1 -14248.321,E2 -14248.321} C_VEL
LIN {X 0,Y 340.696,Z 406.669,A -85,B 0,C 180,E1 -14251.045,E2 -14251.045} C_VEL
LIN {X 0,Y 340.711,Z 406.666,A -85,B 0,C 180,E1 -14255.28,E2 -14255.28} C_VEL
LIN {X 0,Y 340.704,Z 406.669,A -85,B 0,C 180,E1 -14258.388,E2 -14258.388} C_VEL
LIN {X 0,Y 340.694,Z 406.67,A -85,B 0,C 180,E1 -14262.047,E2 -14262.047} C_VEL
LIN {X 0,Y 340.684,Z 406.668,A -85,B 0,C 180,E1 -14265.464,E2 -14265.464} C_VEL
LIN {X 0,Y 340.7,Z 406.671,A -85,B 0,C 180,E1 -14268.695,E2 -14268.695} C_VEL
LIN {X 0,Y 340.738,Z 406.663,A -85,B 0,C 180,E1 -14271.775,E2 -14271.775} C_VEL
LIN {X 0,Y 340.72,Z 406.665,A -85,B 0,C 180,E1 -14275.597,E2 -14275.597} C_VEL
LIN {X 0,Y 340.701,Z 406.668,A -85,B 0,C 180,E1 -14278.958,E2 -14278.958} C_VEL
LIN {X 0,Y 340.727,Z 406.665,A -85,B 0,C 180,E1 -14281.681,E2 -14281.681} C_VEL
LIN {X 0,Y 340.772,Z 406.665,A -85,B 0,C 180,E1 -14284.337,E2 -14284.337} C_VEL
LIN {X 0,Y 340.741,Z 406.669,A -85,B 0,C 180,E1 -14288.208,E2 -14288.208} C_VEL
LIN {X 0,Y 340.824,Z 406.646,A -85,B 0,C 180,E1 -14292.247,E2 -14292.247} C_VEL
LIN {X 0,Y 345.41,Z 419.419,A -85,B 0,C 180,E1 -14293.001,E2 -14293.001} C_VEL
LIN {X 0,Y 348.405,Z 428.687,A -85,B 0,C 180,E1 -14293.684,E2 -14293.684} C_VEL
LIN {X 0,Y 348.501,Z 432.715,A -85,B 0,C 180,E1 -14293.947,E2 -14293.947} C_VEL
LIN {X 0,Y 347.779,Z 445.436,A -85,B 0,C 180,E1 -14294.921,E2 -14294.921} C_VEL
LIN {X 0,Y 347.037,Z 455.727,A -85,B 0,C 180,E1 -14295.937,E2 -14295.937} C_VEL
LIN {X 0,Y 346.037,Z 466.294,A -85,B 0,C 180,E1 -14297.239,E2 -14297.239} C_VEL
LIN {X 0,Y 344.888,Z 476.622,A -85,B 0,C 180,E1 -14298.839,E2 -14298.839} C_VEL
LIN {X 0,Y 344.026,Z 484.224,A -85,B 0,C 180,E1 -14300.299,E2 -14300.299} C_VEL
LIN {X 0,Y 343.071,Z 491.672,A -85,B 0,C 180,E1 -14302.053,E2 -14302.053} C_VEL
LIN {X 0,Y 342.471,Z 496.739,A -85,B 0,C 180,E1 -14303.521,E2 -14303.521} C_VEL
LIN {X 0,Y 341.919,Z 501.642,A -85,B 0,C 180,E1 -14305.285,E2 -14305.285} C_VEL
LIN {X 0,Y 341.427,Z 505.443,A -85,B 0,C 180,E1 -14307.052,E2 -14307.052} C_VEL
LIN {X 0,Y 341.034,Z 508.25,A -85,B 0,C 180,E1 -14308.82,E2 -14308.82} C_VEL
LIN {X 0,Y 340.879,Z 510.505,A -85,B 0,C 180,E1 -14311.183,E2 -14311.183} C_VEL
LIN {X 0,Y 340.804,Z 511.083,A -85,B 0,C 180,E1 -14312.365,E2 -14312.365} C_VEL
LIN {X 0,Y 340.669,Z 511.277,A -85,B 0,C 180,E1 -14313.55,E2 -14313.55} C_VEL
LIN {X 0,Y 341.04,Z 510.415,A -85,B 0,C 180,E1 -14315.915,E2 -14315.915} C_VEL
LIN {X 0,Y 341.392,Z 509.412,A -85,B 0,C 180,E1 -14317.096,E2 -14317.096} C_VEL
LIN {X 0,Y 341.892,Z 506.357,A -85,B 0,C 180,E1 -14319.353,E2 -14319.353} C_VEL
LIN {X 0,Y 342.601,Z 502.572,A -85,B 0,C 180,E1 -14321.239,E2 -14321.239} C_VEL
LIN {X 0,Y 343.263,Z 497.897,A -85,B 0,C 180,E1 -14323.017,E2 -14323.017} C_VEL
LIN {X 0,Y 344.136,Z 491.966,A -85,B 0,C 180,E1 -14324.791,E2 -14324.791} C_VEL
LIN {X 0,Y 345.21,Z 484.511,A -85,B 0,C 180,E1 -14326.561,E2 -14326.561} C_VEL
LIN {X 0,Y 346.555,Z 475.119,A -85,B 0,C 180,E1 -14328.322,E2 -14328.322} C_VEL
LIN {X 0,Y 347.689,Z 465.374,A -85,B 0,C 180,E1 -14329.791,E2 -14329.791} C_VEL
LIN {X 0,Y 348.774,Z 454.339,A -85,B 0,C 180,E1 -14331.113,E2 -14331.113} C_VEL
LIN {X 0,Y 349.68,Z 442.918,A -85,B 0,C 180,E1 -14332.193,E2 -14332.193} C_VEL
LIN {X 0,Y 350.326,Z 433.228,A -85,B 0,C 180,E1 -14332.905,E2 -14332.905} C_VEL
LIN {X 0,Y 349.692,Z 430.203,A -85,B 0,C 180,E1 -14333.15,E2 -14333.15} C_VEL
LIN {X 0,Y 345.663,Z 418.781,A -85,B 0,C 180,E1 -14334.07,E2 -14334.07} C_VEL
LIN {X 0,Y 340.884,Z 407.222,A -85,B 0,C 180,E1 -14334.84,E2 -14334.84} C_VEL
LIN {X 0,Y 340.776,Z 406.656,A -85,B 0,C 180,E1 -14334.903,E2 -14334.903} C_VEL
LIN {X 0,Y 340.747,Z 406.665,A -85,B 0,C 180,E1 -14338.32,E2 -14338.32} C_VEL
LIN {X 0,Y 340.71,Z 406.673,A -85,B 0,C 180,E1 -14341.045,E2 -14341.045} C_VEL
LIN {X 0,Y 340.724,Z 406.671,A -85,B 0,C 180,E1 -14345.279,E2 -14345.279} C_VEL
LIN {X 0,Y 340.715,Z 406.655,A -85,B 0,C 180,E1 -14348.386,E2 -14348.386} C_VEL
LIN {X 0,Y 340.705,Z 406.669,A -85,B 0,C 180,E1 -14352.046,E2 -14352.046} C_VEL
LIN {X 0,Y 340.662,Z 406.672,A -85,B 0,C 180,E1 -14356.226,E2 -14356.226} C_VEL
LIN {X 0,Y 340.661,Z 406.672,A -85,B 0,C 180,E1 -14356.485,E2 -14356.485} C_VEL
LIN {X 0,Y 340.009,Z 406.757,A -85,B 0,C 180,E1 -14357.471,E2 -14357.471} C_VEL
LIN {X 0,Y 337.17,Z 407.103,A -85,B 0,C 180,E1 -14359.076,E2 -14359.076} C_VEL
LIN {X 0,Y 334.758,Z 407.386,A -85,B 0,C 180,E1 -14360.375,E2 -14360.375} C_VEL
LIN {X 0,Y 333.725,Z 407.508,A -85,B 0,C 180,E1 -14361.381,E2 -14361.381} C_VEL
LIN {X 0,Y 333.642,Z 407.519,A -85,B 0,C 180,E1 -14361.721,E2 -14361.721} C_VEL
LIN {X 0,Y 333.68,Z 407.545,A -85,B 0,C 180,E1 -14365.341,E2 -14365.341} C_VEL
LIN {X 0,Y 333.696,Z 407.504,A -85,B 0,C 180,E1 -14369.637,E2 -14369.637} C_VEL
LIN {X 0,Y 333.745,Z 407.514,A -85,B 0,C 180,E1 -14372.401,E2 -14372.401} C_VEL
LIN {X 0,Y 333.731,Z 407.537,A -85,B 0,C 180,E1 -14375.091,E2 -14375.091} C_VEL
LIN {X 0,Y 333.695,Z 407.571,A -85,B 0,C 180,E1 -14378.129,E2 -14378.129} C_VEL
LIN {X 0,Y 337.844,Z 421.589,A -85,B 0,C 180,E1 -14379.41,E2 -14379.41} C_VEL
LIN {X 0,Y 340.807,Z 431.969,A -85,B 0,C 180,E1 -14380.516,E2 -14380.516} C_VEL
LIN {X 0,Y 339.714,Z 445.113,A -85,B 0,C 180,E1 -14381.921,E2 -14381.921} C_VEL
LIN {X 0,Y 338.514,Z 457.766,A -85,B 0,C 180,E1 -14383.568,E2 -14383.568} C_VEL
LIN {X 0,Y 337.384,Z 468.251,A -85,B 0,C 180,E1 -14385.216,E2 -14385.216} C_VEL
LIN {X 0,Y 336.471,Z 477.828,A -85,B 0,C 180,E1 -14387.024,E2 -14387.024} C_VEL
LIN {X 0,Y 335.517,Z 487.07,A -85,B 0,C 180,E1 -14389.133,E2 -14389.133} C_VEL
LIN {X 0,Y 334.855,Z 494.318,A -85,B 0,C 180,E1 -14391.147,E2 -14391.147} C_VEL
LIN {X 0,Y 334.385,Z 500.759,A -85,B 0,C 180,E1 -14393.362,E2 -14393.362} C_VEL
LIN {X 0,Y 333.855,Z 505.001,A -85,B 0,C 180,E1 -14395.169,E2 -14395.169} C_VEL
LIN {X 0,Y 333.68,Z 507.323,A -85,B 0,C 180,E1 -14396.377,E2 -14396.377} C_VEL
LIN {X 0,Y 333.871,Z 510.842,A -85,B 0,C 180,E1 -14398.794,E2 -14398.794} C_VEL
LIN {X 0,Y 333.955,Z 513.031,A -85,B 0,C 180,E1 -14401.206,E2 -14401.206} C_VEL
LIN {X 0,Y 334.335,Z 513.865,A -85,B 0,C 180,E1 -14403.615,E2 -14403.615} C_VEL
LIN {X 0,Y 334.905,Z 513.36,A -85,B 0,C 180,E1 -14406.023,E2 -14406.023} C_VEL
LIN {X 0,Y 335.797,Z 511.506,A -85,B 0,C 180,E1 -14408.424,E2 -14408.424} C_VEL
LIN {X 0,Y 337.039,Z 508.272,A -85,B 0,C 180,E1 -14410.817,E2 -14410.817} C_VEL
LIN {X 0,Y 338.516,Z 503.615,A -85,B 0,C 180,E1 -14413.201,E2 -14413.201} C_VEL
LIN {X 0,Y 339.917,Z 499.077,A -85,B 0,C 180,E1 -14414.978,E2 -14414.978} C_VEL
LIN {X 0,Y 342.155,Z 491.49,A -85,B 0,C 180,E1 -14417.327,E2 -14417.327} C_VEL
LIN {X 0,Y 344.408,Z 483.312,A -85,B 0,C 180,E1 -14419.329,E2 -14419.329} C_VEL
LIN {X 0,Y 347.025,Z 472.911,A -85,B 0,C 180,E1 -14421.379,E2 -14421.379} C_VEL
LIN {X 0,Y 349.442,Z 462.318,A -85,B 0,C 180,E1 -14423.09,E2 -14423.09} C_VEL
LIN {X 0,Y 351.912,Z 450.506,A -85,B 0,C 180,E1 -14424.638,E2 -14424.638} C_VEL
LIN {X 0,Y 352.522,Z 447.449,A -85,B 0,C 180,E1 -14424.993,E2 -14424.993} C_VEL
LIN {X 0,Y 350.5,Z 439.48,A -85,B 0,C 180,E1 -14426.444,E2 -14426.444} C_VEL
LIN {X 0,Y 347.033,Z 430.624,A -85,B 0,C 180,E1 -14428.231,E2 -14428.231} C_VEL
LIN {X 0,Y 342.803,Z 422.087,A -85,B 0,C 180,E1 -14430.164,E2 -14430.164} C_VEL
LIN {X 0,Y 339.861,Z 417.512,A -85,B 0,C 180,E1 -14431.415,E2 -14431.415} C_VEL
LIN {X 0,Y 337.094,Z 414.707,A -85,B 0,C 180,E1 -14432.511,E2 -14432.511} C_VEL
LIN {X 0,Y 335.591,Z 413.535,A -85,B 0,C 180,E1 -14433.102,E2 -14433.102} C_VEL
LIN {X 0,Y 334.62,Z 411.76,A -85,B 0,C 180,E1 -14433.638,E2 -14433.638} C_VEL
LIN {X 0,Y 335.24,Z 414.736,A -85,B 0,C 180,E1 -14437.442,E2 -14437.442} C_VEL
LIN {X 0,Y 335.921,Z 417.823,A -85,B 0,C 180,E1 -14440.434,E2 -14440.434} C_VEL
LIN {X 0,Y 336.761,Z 421.792,A -85,B 0,C 180,E1 -14443.526,E2 -14443.526} C_VEL
LIN {X 0,Y 337.762,Z 426.796,A -85,B 0,C 180,E1 -14446.741,E2 -14446.741} C_VEL
LIN {X 0,Y 338.443,Z 431.238,A -85,B 0,C 180,E1 -14449.183,E2 -14449.183} C_VEL
LIN {X 0,Y 338.155,Z 433.541,A -85,B 0,C 180,E1 -14450.263,E2 -14450.263} C_VEL
LIN {X 0,Y 336.209,Z 443.835,A -85,B 0,C 180,E1 -14454.611,E2 -14454.611} C_VEL
LIN {X 0,Y 335.365,Z 450.939,A -85,B 0,C 180,E1 -14457.344,E2 -14457.344} C_VEL
LIN {X 0,Y 336.437,Z 455.777,A -85,B 0,C 180,E1 -14457.971,E2 -14457.971} C_VEL
LIN {X 0,Y 337.427,Z 458.8,A -85,B 0,C 180,E1 -14458.425,E2 -14458.425} C_VEL
LIN {X 0,Y 339.165,Z 465.916,A -85,B 0,C 180,E1 -14459.331,E2 -14459.331} C_VEL
LIN {X 0,Y 342.055,Z 479.88,A -85,B 0,C 180,E1 -14460.987,E2 -14460.987} C_VEL
LIN {X 0,Y 343.832,Z 494.647,A -85,B 0,C 180,E1 -14462.586,E2 -14462.586} C_VEL
LIN {X 0,Y 344.258,Z 508.211,A -85,B 0,C 180,E1 -14464.009,E2 -14464.009} C_VEL
LIN {X 0,Y 343.449,Z 520.895,A -85,B 0,C 180,E1 -14465.358,E2 -14465.358} C_VEL
LIN {X 0,Y 342.055,Z 534.876,A -85,B 0,C 180,E1 -14467.021,E2 -14467.021} C_VEL
LIN {X 0,Y 340.172,Z 545.573,A -85,B 0,C 180,E1 -14468.424,E2 -14468.424} C_VEL
LIN {X 0,Y 338.139,Z 555.669,A -85,B 0,C 180,E1 -14469.943,E2 -14469.943} C_VEL
LIN {X 0,Y 335.995,Z 567.357,A -85,B 0,C 180,E1 -14472.028,E2 -14472.028} C_VEL
LIN {X 0,Y 334.494,Z 577.173,A -85,B 0,C 180,E1 -14474.148,E2 -14474.148} C_VEL
LIN {X 0,Y 333.422,Z 585.354,A -85,B 0,C 180,E1 -14476.265,E2 -14476.265} C_VEL
LIN {X 0,Y 332.904,Z 592.269,A -85,B 0,C 180,E1 -14478.429,E2 -14478.429} C_VEL
LIN {X 0,Y 332.69,Z 598.526,A -85,B 0,C 180,E1 -14480.883,E2 -14480.883} C_VEL
LIN {X 0,Y 332.824,Z 602.615,A -85,B 0,C 180,E1 -14482.961,E2 -14482.961} C_VEL
LIN {X 0,Y 333.11,Z 605.757,A -85,B 0,C 180,E1 -14485.158,E2 -14485.158} C_VEL
LIN {X 0,Y 333.221,Z 606.953,A -85,B 0,C 180,E1 -14486.371,E2 -14486.371} C_VEL
LIN {X 0,Y 333.577,Z 608.239,A -85,B 0,C 180,E1 -14488.791,E2 -14488.791} C_VEL
LIN {X 0,Y 333.771,Z 608.313,A -85,B 0,C 180,E1 -14489.999,E2 -14489.999} C_VEL
LIN {X 0,Y 333.617,Z 607.95,A -85,B 0,C 180,E1 -14491.206,E2 -14491.206} C_VEL
LIN {X 0,Y 333.329,Z 606.073,A -85,B 0,C 180,E1 -14493.625,E2 -14493.625} C_VEL
LIN {X 0,Y 333.257,Z 604.558,A -85,B 0,C 180,E1 -14494.838,E2 -14494.838} C_VEL
LIN {X 0,Y 333.079,Z 600.921,A -85,B 0,C 180,E1 -14496.949,E2 -14496.949} C_VEL
LIN {X 0,Y 332.949,Z 595.847,A -85,B 0,C 180,E1 -14499.108,E2 -14499.108} C_VEL
LIN {X 0,Y 333.089,Z 589.369,A -85,B 0,C 180,E1 -14501.253,E2 -14501.253} C_VEL
LIN {X 0,Y 333.484,Z 581.257,A -85,B 0,C 180,E1 -14503.403,E2 -14503.403} C_VEL
LIN {X 0,Y 334.247,Z 572.788,A -85,B 0,C 180,E1 -14505.236,E2 -14505.236} C_VEL
LIN {X 0,Y 335.216,Z 562.551,A -85,B 0,C 180,E1 -14507.067,E2 -14507.067} C_VEL
LIN {X 0,Y 336.583,Z 551.308,A -85,B 0,C 180,E1 -14508.724,E2 -14508.724} C_VEL
LIN {X 0,Y 337.975,Z 538.916,A -85,B 0,C 180,E1 -14510.223,E2 -14510.223} C_VEL
LIN {X 0,Y 338.748,Z 531.446,A -85,B 0,C 180,E1 -14510.995,E2 -14510.995} C_VEL
LIN {X 0,Y 337.846,Z 517.38,A -85,B 0,C 180,E1 -14512.267,E2 -14512.267} C_VEL
LIN {X 0,Y 336.393,Z 502.09,A -85,B 0,C 180,E1 -14513.386,E2 -14513.386} C_VEL
LIN {X 0,Y 334.835,Z 486.509,A -85,B 0,C 180,E1 -14514.266,E2 -14514.266} C_VEL
LIN {X 0,Y 333.876,Z 476.993,A -85,B 0,C 180,E1 -14514.688,E2 -14514.688} C_VEL
LIN {X 0,Y 334.8,Z 465.196,A -85,B 0,C 180,E1 -14518.867,E2 -14518.867} C_VEL
LIN {X 0,Y 335.976,Z 453.839,A -85,B 0,C 180,E1 -14522.946,E2 -14522.946} C_VEL
LIN {X 0,Y 336.951,Z 446.189,A -85,B 0,C 180,E1 -14525.731,E2 -14525.731} C_VEL
LIN {X 0,Y 338.504,Z 434.53,A -85,B 0,C 180,E1 -14530.06,E2 -14530.06} C_VEL
LIN {X 0,Y 338.279,Z 430.425,A -85,B 0,C 180,E1 -14531.666,E2 -14531.666} C_VEL
LIN {X 0,Y 336.518,Z 421.811,A -85,B 0,C 180,E1 -14535.238,E2 -14535.238} C_VEL
LIN {X 0,Y 334.746,Z 412.952,A -85,B 0,C 180,E1 -14539.094,E2 -14539.094} C_VEL
LIN {X 0,Y 333.673,Z 407.548,A -85,B 0,C 180,E1 -14541.632,E2 -14541.632} C_VEL
LIN {X 0,Y 333.665,Z 407.549,A -85,B 0,C 180,E1 -14545.34,E2 -14545.34} C_VEL
LIN {X 0,Y 333.693,Z 407.541,A -85,B 0,C 180,E1 -14549.709,E2 -14549.709} C_VEL
LIN {X 0,Y 333.735,Z 407.536,A -85,B 0,C 180,E1 -14552.401,E2 -14552.401} C_VEL
LIN {X 0,Y 333.717,Z 407.542,A -85,B 0,C 180,E1 -14555.09,E2 -14555.09} C_VEL
LIN {X 0,Y 333.67,Z 407.548,A -85,B 0,C 180,E1 -14559.019,E2 -14559.019} C_VEL
LIN {X 0,Y 333.783,Z 407.531,A -85,B 0,C 180,E1 -14561.589,E2 -14561.589} C_VEL
LIN {X 0,Y 333.798,Z 407.528,A -85,B 0,C 180,E1 -14565.576,E2 -14565.576} C_VEL
LIN {X 0,Y 333.827,Z 407.527,A -85,B 0,C 180,E1 -14569.078,E2 -14569.078} C_VEL
LIN {X 0,Y 334.015,Z 407.504,A -85,B 0,C 180,E1 -14572.748,E2 -14572.748} C_VEL
LIN {X 0,Y 333.804,Z 407.529,A -85,B 0,C 180,E1 -14575.169,E2 -14575.169} C_VEL
LIN {X 0,Y 334.122,Z 407.488,A -85,B 0,C 180,E1 -14577.589,E2 -14577.589} C_VEL
LIN {X 0,Y 334.257,Z 407.47,A -85,B 0,C 180,E1 -14580,E2 -14580} C_VEL
LIN {X 0,Y 334.122,Z 407.488,A -85,B 0,C 180,E1 -14582.411,E2 -14582.411} C_VEL
LIN {X 0,Y 334.015,Z 407.498,A -85,B 0,C 180,E1 -14587.253,E2 -14587.253} C_VEL
LIN {X 0,Y 333.828,Z 407.527,A -85,B 0,C 180,E1 -14590.922,E2 -14590.922} C_VEL
LIN {X 0,Y 333.799,Z 407.532,A -85,B 0,C 180,E1 -14594.635,E2 -14594.635} C_VEL
LIN {X 0,Y 333.788,Z 407.533,A -85,B 0,C 180,E1 -14598.656,E2 -14598.656} C_VEL
LIN {X 0,Y 333.683,Z 407.543,A -85,B 0,C 180,E1 -14602.279,E2 -14602.279} C_VEL
LIN {X 0,Y 333.727,Z 407.538,A -85,B 0,C 180,E1 -14606.247,E2 -14606.247} C_VEL
LIN {X 0,Y 333.703,Z 407.536,A -85,B 0,C 180,E1 -14608.973,E2 -14608.973} C_VEL
LIN {X 0,Y 333.636,Z 407.551,A -85,B 0,C 180,E1 -14612.588,E2 -14612.588} C_VEL
LIN {X 0,Y 333.67,Z 407.544,A -85,B 0,C 180,E1 -14616.14,E2 -14616.14} C_VEL
LIN {X 0,Y 333.641,Z 407.546,A -85,B 0,C 180,E1 -14619.194,E2 -14619.194} C_VEL
LIN {X 0,Y 333.629,Z 407.554,A -85,B 0,C 180,E1 -14622.502,E2 -14622.502} C_VEL
LIN {X 0,Y 333.627,Z 407.547,A -85,B 0,C 180,E1 -14625.963,E2 -14625.963} C_VEL
LIN {X 0,Y 333.652,Z 407.546,A -85,B 0,C 180,E1 -14629.315,E2 -14629.315} C_VEL
LIN {X 0,Y 333.654,Z 407.549,A -85,B 0,C 180,E1 -14632.351,E2 -14632.351} C_VEL
LIN {X 0,Y 333.672,Z 407.543,A -85,B 0,C 180,E1 -14635.343,E2 -14635.343} C_VEL
LIN {X 0,Y 333.702,Z 407.539,A -85,B 0,C 180,E1 -14639.711,E2 -14639.711} C_VEL
LIN {X 0,Y 333.734,Z 407.537,A -85,B 0,C 180,E1 -14643.755,E2 -14643.755} C_VEL
LIN {X 0,Y 333.72,Z 407.541,A -85,B 0,C 180,E1 -14647.916,E2 -14647.916} C_VEL
LIN {X 0,Y 333.795,Z 407.522,A -85,B 0,C 180,E1 -14651.817,E2 -14651.817} C_VEL
LIN {X 0,Y 336.18,Z 414.134,A -85,B 0,C 180,E1 -14652.188,E2 -14652.188} C_VEL
LIN {X 0,Y 340.643,Z 426.837,A -85,B 0,C 180,E1 -14653.077,E2 -14653.077} C_VEL
LIN {X 0,Y 341.933,Z 431.479,A -85,B 0,C 180,E1 -14653.447,E2 -14653.447} C_VEL
LIN {X 0,Y 341.212,Z 443.975,A -85,B 0,C 180,E1 -14654.361,E2 -14654.361} C_VEL
LIN {X 0,Y 340.374,Z 455.697,A -85,B 0,C 180,E1 -14655.503,E2 -14655.503} C_VEL
LIN {X 0,Y 339.329,Z 466.527,A -85,B 0,C 180,E1 -14656.832,E2 -14656.832} C_VEL
LIN {X 0,Y 338.236,Z 476.121,A -85,B 0,C 180,E1 -14658.313,E2 -14658.313} C_VEL
LIN {X 0,Y 337.3,Z 483.976,A -85,B 0,C 180,E1 -14659.8,E2 -14659.8} C_VEL
LIN {X 0,Y 336.234,Z 491.69,A -85,B 0,C 180,E1 -14661.588,E2 -14661.588} C_VEL
LIN {X 0,Y 335.504,Z 497.855,A -85,B 0,C 180,E1 -14663.386,E2 -14663.386} C_VEL
